(* IEC 61131-3 sources: AXOpen/src/components.cognex.vision/app/SystemConstants (part 2) *)

(* ---- plc_main_IoAddresses.st ---- *)
CONFIGURATION IoAddresses
    VAR_GLOBAL
        CommunicationCard_Engine_Control_1_InputAddress AT %IL1288: LWORD;
        CommunicationCard_Engine_Control_1_OutputAddress AT %QB1267: BYTE;
        CommunicationCard_Engine_Control_2_InputAddress AT %IL1280: LWORD;
        CommunicationCard_Engine_Control_2_OutputAddress AT %QB1266: BYTE;
        CommunicationCard_Engine_Control_3_InputAddress AT %IL1272: LWORD;
        CommunicationCard_Engine_Control_3_OutputAddress AT %QB1265: BYTE;
        CommunicationCard_Engine_Control_4_InputAddress AT %IL1264: LWORD;
        CommunicationCard_Engine_Control_4_OutputAddress AT %QB1264: BYTE;
        CommunicationCard_Result_Data_240_bytes_1_InputAddress_0 AT %IL1024: LWORD;
        CommunicationCard_Result_Data_240_bytes_1_InputAddress_1 AT %IL1032: LWORD;
        CommunicationCard_Result_Data_240_bytes_1_InputAddress_2 AT %IL1040: LWORD;
        CommunicationCard_Result_Data_240_bytes_1_InputAddress_3 AT %IL1048: LWORD;
        CommunicationCard_Result_Data_240_bytes_1_InputAddress_4 AT %IL1056: LWORD;
        CommunicationCard_Result_Data_240_bytes_1_InputAddress_5 AT %IL1064: LWORD;
        CommunicationCard_Result_Data_240_bytes_1_InputAddress_6 AT %IL1072: LWORD;
        CommunicationCard_Result_Data_240_bytes_1_InputAddress_7 AT %IL1080: LWORD;
        CommunicationCard_Result_Data_240_bytes_1_InputAddress_8 AT %IL1088: LWORD;
        CommunicationCard_Result_Data_240_bytes_1_InputAddress_9 AT %IL1096: LWORD;
        CommunicationCard_Result_Data_240_bytes_1_InputAddress_10 AT %IL1104: LWORD;
        CommunicationCard_Result_Data_240_bytes_1_InputAddress_11 AT %IL1112: LWORD;
        CommunicationCard_Result_Data_240_bytes_1_InputAddress_12 AT %IL1120: LWORD;
        CommunicationCard_Result_Data_240_bytes_1_InputAddress_13 AT %IL1128: LWORD;
        CommunicationCard_Result_Data_240_bytes_1_InputAddress_14 AT %IL1136: LWORD;
        CommunicationCard_Result_Data_240_bytes_1_InputAddress_15 AT %IL1144: LWORD;
        CommunicationCard_Result_Data_240_bytes_1_InputAddress_16 AT %IL1152: LWORD;
        CommunicationCard_Result_Data_240_bytes_1_InputAddress_17 AT %IL1160: LWORD;
        CommunicationCard_Result_Data_240_bytes_1_InputAddress_18 AT %IL1168: LWORD;
        CommunicationCard_Result_Data_240_bytes_1_InputAddress_19 AT %IL1176: LWORD;
        CommunicationCard_Result_Data_240_bytes_1_InputAddress_20 AT %IL1184: LWORD;
        CommunicationCard_Result_Data_240_bytes_1_InputAddress_21 AT %IL1192: LWORD;
        CommunicationCard_Result_Data_240_bytes_1_InputAddress_22 AT %IL1200: LWORD;
        CommunicationCard_Result_Data_240_bytes_1_InputAddress_23 AT %IL1208: LWORD;
        CommunicationCard_Result_Data_240_bytes_1_InputAddress_24 AT %IL1216: LWORD;
        CommunicationCard_Result_Data_240_bytes_1_InputAddress_25 AT %IL1224: LWORD;
        CommunicationCard_Result_Data_240_bytes_1_InputAddress_26 AT %IL1232: LWORD;
        CommunicationCard_Result_Data_240_bytes_1_InputAddress_27 AT %IL1240: LWORD;
        CommunicationCard_Result_Data_240_bytes_1_InputAddress_28 AT %IL1248: LWORD;
        CommunicationCard_Result_Data_240_bytes_1_InputAddress_29 AT %IL1256: LWORD;
        CommunicationCard_Result_Data_240_bytes_2_InputAddress_0 AT %IL784: LWORD;
        CommunicationCard_Result_Data_240_bytes_2_InputAddress_1 AT %IL792: LWORD;
        CommunicationCard_Result_Data_240_bytes_2_InputAddress_2 AT %IL800: LWORD;
        CommunicationCard_Result_Data_240_bytes_2_InputAddress_3 AT %IL808: LWORD;
        CommunicationCard_Result_Data_240_bytes_2_InputAddress_4 AT %IL816: LWORD;
        CommunicationCard_Result_Data_240_bytes_2_InputAddress_5 AT %IL824: LWORD;
        CommunicationCard_Result_Data_240_bytes_2_InputAddress_6 AT %IL832: LWORD;
        CommunicationCard_Result_Data_240_bytes_2_InputAddress_7 AT %IL840: LWORD;
        CommunicationCard_Result_Data_240_bytes_2_InputAddress_8 AT %IL848: LWORD;
        CommunicationCard_Result_Data_240_bytes_2_InputAddress_9 AT %IL856: LWORD;
        CommunicationCard_Result_Data_240_bytes_2_InputAddress_10 AT %IL864: LWORD;
        CommunicationCard_Result_Data_240_bytes_2_InputAddress_11 AT %IL872: LWORD;
        CommunicationCard_Result_Data_240_bytes_2_InputAddress_12 AT %IL880: LWORD;
        CommunicationCard_Result_Data_240_bytes_2_InputAddress_13 AT %IL888: LWORD;
        CommunicationCard_Result_Data_240_bytes_2_InputAddress_14 AT %IL896: LWORD;
        CommunicationCard_Result_Data_240_bytes_2_InputAddress_15 AT %IL904: LWORD;
        CommunicationCard_Result_Data_240_bytes_2_InputAddress_16 AT %IL912: LWORD;
        CommunicationCard_Result_Data_240_bytes_2_InputAddress_17 AT %IL920: LWORD;
        CommunicationCard_Result_Data_240_bytes_2_InputAddress_18 AT %IL928: LWORD;
        CommunicationCard_Result_Data_240_bytes_2_InputAddress_19 AT %IL936: LWORD;
        CommunicationCard_Result_Data_240_bytes_2_InputAddress_20 AT %IL944: LWORD;
        CommunicationCard_Result_Data_240_bytes_2_InputAddress_21 AT %IL952: LWORD;
        CommunicationCard_Result_Data_240_bytes_2_InputAddress_22 AT %IL960: LWORD;
        CommunicationCard_Result_Data_240_bytes_2_InputAddress_23 AT %IL968: LWORD;
        CommunicationCard_Result_Data_240_bytes_2_InputAddress_24 AT %IL976: LWORD;
        CommunicationCard_Result_Data_240_bytes_2_InputAddress_25 AT %IL984: LWORD;
        CommunicationCard_Result_Data_240_bytes_2_InputAddress_26 AT %IL992: LWORD;
        CommunicationCard_Result_Data_240_bytes_2_InputAddress_27 AT %IL1000: LWORD;
        CommunicationCard_Result_Data_240_bytes_2_InputAddress_28 AT %IL1008: LWORD;
        CommunicationCard_Result_Data_240_bytes_2_InputAddress_29 AT %IL1016: LWORD;
        CommunicationCard_Result_Data_240_bytes_3_InputAddress_0 AT %IL544: LWORD;
        CommunicationCard_Result_Data_240_bytes_3_InputAddress_1 AT %IL552: LWORD;
        CommunicationCard_Result_Data_240_bytes_3_InputAddress_2 AT %IL560: LWORD;
        CommunicationCard_Result_Data_240_bytes_3_InputAddress_3 AT %IL568: LWORD;
        CommunicationCard_Result_Data_240_bytes_3_InputAddress_4 AT %IL576: LWORD;
        CommunicationCard_Result_Data_240_bytes_3_InputAddress_5 AT %IL584: LWORD;
        CommunicationCard_Result_Data_240_bytes_3_InputAddress_6 AT %IL592: LWORD;
        CommunicationCard_Result_Data_240_bytes_3_InputAddress_7 AT %IL600: LWORD;
        CommunicationCard_Result_Data_240_bytes_3_InputAddress_8 AT %IL608: LWORD;
        CommunicationCard_Result_Data_240_bytes_3_InputAddress_9 AT %IL616: LWORD;
        CommunicationCard_Result_Data_240_bytes_3_InputAddress_10 AT %IL624: LWORD;
        CommunicationCard_Result_Data_240_bytes_3_InputAddress_11 AT %IL632: LWORD;
        CommunicationCard_Result_Data_240_bytes_3_InputAddress_12 AT %IL640: LWORD;
        CommunicationCard_Result_Data_240_bytes_3_InputAddress_13 AT %IL648: LWORD;
        CommunicationCard_Result_Data_240_bytes_3_InputAddress_14 AT %IL656: LWORD;
        CommunicationCard_Result_Data_240_bytes_3_InputAddress_15 AT %IL664: LWORD;
        CommunicationCard_Result_Data_240_bytes_3_InputAddress_16 AT %IL672: LWORD;
        CommunicationCard_Result_Data_240_bytes_3_InputAddress_17 AT %IL680: LWORD;
        CommunicationCard_Result_Data_240_bytes_3_InputAddress_18 AT %IL688: LWORD;
        CommunicationCard_Result_Data_240_bytes_3_InputAddress_19 AT %IL696: LWORD;
        CommunicationCard_Result_Data_240_bytes_3_InputAddress_20 AT %IL704: LWORD;
        CommunicationCard_Result_Data_240_bytes_3_InputAddress_21 AT %IL712: LWORD;
        CommunicationCard_Result_Data_240_bytes_3_InputAddress_22 AT %IL720: LWORD;
        CommunicationCard_Result_Data_240_bytes_3_InputAddress_23 AT %IL728: LWORD;
        CommunicationCard_Result_Data_240_bytes_3_InputAddress_24 AT %IL736: LWORD;
        CommunicationCard_Result_Data_240_bytes_3_InputAddress_25 AT %IL744: LWORD;
        CommunicationCard_Result_Data_240_bytes_3_InputAddress_26 AT %IL752: LWORD;
        CommunicationCard_Result_Data_240_bytes_3_InputAddress_27 AT %IL760: LWORD;
        CommunicationCard_Result_Data_240_bytes_3_InputAddress_28 AT %IL768: LWORD;
        CommunicationCard_Result_Data_240_bytes_3_InputAddress_29 AT %IL776: LWORD;
        CommunicationCard_Result_Data_240_bytes_4_InputAddress_0 AT %IL304: LWORD;
        CommunicationCard_Result_Data_240_bytes_4_InputAddress_1 AT %IL312: LWORD;
        CommunicationCard_Result_Data_240_bytes_4_InputAddress_2 AT %IL320: LWORD;
        CommunicationCard_Result_Data_240_bytes_4_InputAddress_3 AT %IL328: LWORD;
        CommunicationCard_Result_Data_240_bytes_4_InputAddress_4 AT %IL336: LWORD;
        CommunicationCard_Result_Data_240_bytes_4_InputAddress_5 AT %IL344: LWORD;
        CommunicationCard_Result_Data_240_bytes_4_InputAddress_6 AT %IL352: LWORD;
        CommunicationCard_Result_Data_240_bytes_4_InputAddress_7 AT %IL360: LWORD;
        CommunicationCard_Result_Data_240_bytes_4_InputAddress_8 AT %IL368: LWORD;
        CommunicationCard_Result_Data_240_bytes_4_InputAddress_9 AT %IL376: LWORD;
        CommunicationCard_Result_Data_240_bytes_4_InputAddress_10 AT %IL384: LWORD;
        CommunicationCard_Result_Data_240_bytes_4_InputAddress_11 AT %IL392: LWORD;
        CommunicationCard_Result_Data_240_bytes_4_InputAddress_12 AT %IL400: LWORD;
        CommunicationCard_Result_Data_240_bytes_4_InputAddress_13 AT %IL408: LWORD;
        CommunicationCard_Result_Data_240_bytes_4_InputAddress_14 AT %IL416: LWORD;
        CommunicationCard_Result_Data_240_bytes_4_InputAddress_15 AT %IL424: LWORD;
        CommunicationCard_Result_Data_240_bytes_4_InputAddress_16 AT %IL432: LWORD;
        CommunicationCard_Result_Data_240_bytes_4_InputAddress_17 AT %IL440: LWORD;
        CommunicationCard_Result_Data_240_bytes_4_InputAddress_18 AT %IL448: LWORD;
        CommunicationCard_Result_Data_240_bytes_4_InputAddress_19 AT %IL456: LWORD;
        CommunicationCard_Result_Data_240_bytes_4_InputAddress_20 AT %IL464: LWORD;
        CommunicationCard_Result_Data_240_bytes_4_InputAddress_21 AT %IL472: LWORD;
        CommunicationCard_Result_Data_240_bytes_4_InputAddress_22 AT %IL480: LWORD;
        CommunicationCard_Result_Data_240_bytes_4_InputAddress_23 AT %IL488: LWORD;
        CommunicationCard_Result_Data_240_bytes_4_InputAddress_24 AT %IL496: LWORD;
        CommunicationCard_Result_Data_240_bytes_4_InputAddress_25 AT %IL504: LWORD;
        CommunicationCard_Result_Data_240_bytes_4_InputAddress_26 AT %IL512: LWORD;
        CommunicationCard_Result_Data_240_bytes_4_InputAddress_27 AT %IL520: LWORD;
        CommunicationCard_Result_Data_240_bytes_4_InputAddress_28 AT %IL528: LWORD;
        CommunicationCard_Result_Data_240_bytes_4_InputAddress_29 AT %IL536: LWORD;
        CommunicationCard_Result_Data_240_bytes_5_InputAddress_0 AT %IL64: LWORD;
        CommunicationCard_Result_Data_240_bytes_5_InputAddress_1 AT %IL72: LWORD;
        CommunicationCard_Result_Data_240_bytes_5_InputAddress_2 AT %IL80: LWORD;
        CommunicationCard_Result_Data_240_bytes_5_InputAddress_3 AT %IL88: LWORD;
        CommunicationCard_Result_Data_240_bytes_5_InputAddress_4 AT %IL96: LWORD;
        CommunicationCard_Result_Data_240_bytes_5_InputAddress_5 AT %IL104: LWORD;
        CommunicationCard_Result_Data_240_bytes_5_InputAddress_6 AT %IL112: LWORD;
        CommunicationCard_Result_Data_240_bytes_5_InputAddress_7 AT %IL120: LWORD;
        CommunicationCard_Result_Data_240_bytes_5_InputAddress_8 AT %IL128: LWORD;
        CommunicationCard_Result_Data_240_bytes_5_InputAddress_9 AT %IL136: LWORD;
        CommunicationCard_Result_Data_240_bytes_5_InputAddress_10 AT %IL144: LWORD;
        CommunicationCard_Result_Data_240_bytes_5_InputAddress_11 AT %IL152: LWORD;
        CommunicationCard_Result_Data_240_bytes_5_InputAddress_12 AT %IL160: LWORD;
        CommunicationCard_Result_Data_240_bytes_5_InputAddress_13 AT %IL168: LWORD;
        CommunicationCard_Result_Data_240_bytes_5_InputAddress_14 AT %IL176: LWORD;
        CommunicationCard_Result_Data_240_bytes_5_InputAddress_15 AT %IL184: LWORD;
        CommunicationCard_Result_Data_240_bytes_5_InputAddress_16 AT %IL192: LWORD;
        CommunicationCard_Result_Data_240_bytes_5_InputAddress_17 AT %IL200: LWORD;
        CommunicationCard_Result_Data_240_bytes_5_InputAddress_18 AT %IL208: LWORD;
        CommunicationCard_Result_Data_240_bytes_5_InputAddress_19 AT %IL216: LWORD;
        CommunicationCard_Result_Data_240_bytes_5_InputAddress_20 AT %IL224: LWORD;
        CommunicationCard_Result_Data_240_bytes_5_InputAddress_21 AT %IL232: LWORD;
        CommunicationCard_Result_Data_240_bytes_5_InputAddress_22 AT %IL240: LWORD;
        CommunicationCard_Result_Data_240_bytes_5_InputAddress_23 AT %IL248: LWORD;
        CommunicationCard_Result_Data_240_bytes_5_InputAddress_24 AT %IL256: LWORD;
        CommunicationCard_Result_Data_240_bytes_5_InputAddress_25 AT %IL264: LWORD;
        CommunicationCard_Result_Data_240_bytes_5_InputAddress_26 AT %IL272: LWORD;
        CommunicationCard_Result_Data_240_bytes_5_InputAddress_27 AT %IL280: LWORD;
        CommunicationCard_Result_Data_240_bytes_5_InputAddress_28 AT %IL288: LWORD;
        CommunicationCard_Result_Data_240_bytes_5_InputAddress_29 AT %IL296: LWORD;
        CommunicationCard_Result_Data_64_bytes_1_InputAddress_0 AT %IL0: LWORD;
        CommunicationCard_Result_Data_64_bytes_1_InputAddress_1 AT %IL8: LWORD;
        CommunicationCard_Result_Data_64_bytes_1_InputAddress_2 AT %IL16: LWORD;
        CommunicationCard_Result_Data_64_bytes_1_InputAddress_3 AT %IL24: LWORD;
        CommunicationCard_Result_Data_64_bytes_1_InputAddress_4 AT %IL32: LWORD;
        CommunicationCard_Result_Data_64_bytes_1_InputAddress_5 AT %IL40: LWORD;
        CommunicationCard_Result_Data_64_bytes_1_InputAddress_6 AT %IL48: LWORD;
        CommunicationCard_Result_Data_64_bytes_1_InputAddress_7 AT %IL56: LWORD;
        CommunicationCard_System_Control_InputAddress_0 AT %IL1296: LWORD;
        CommunicationCard_System_Control_InputAddress_1 AT %IL1304: LWORD;
        CommunicationCard_System_Control_OutputAddress_0 AT %QL1268: LWORD;
        CommunicationCard_System_Control_OutputAddress_1 AT %QL1276: LWORD;
        CommunicationCard_User_Data_240_bytes_1_OutputAddress_0 AT %QL1024: LWORD;
        CommunicationCard_User_Data_240_bytes_1_OutputAddress_1 AT %QL1032: LWORD;
        CommunicationCard_User_Data_240_bytes_1_OutputAddress_2 AT %QL1040: LWORD;
        CommunicationCard_User_Data_240_bytes_1_OutputAddress_3 AT %QL1048: LWORD;
        CommunicationCard_User_Data_240_bytes_1_OutputAddress_4 AT %QL1056: LWORD;
        CommunicationCard_User_Data_240_bytes_1_OutputAddress_5 AT %QL1064: LWORD;
        CommunicationCard_User_Data_240_bytes_1_OutputAddress_6 AT %QL1072: LWORD;
        CommunicationCard_User_Data_240_bytes_1_OutputAddress_7 AT %QL1080: LWORD;
        CommunicationCard_User_Data_240_bytes_1_OutputAddress_8 AT %QL1088: LWORD;
        CommunicationCard_User_Data_240_bytes_1_OutputAddress_9 AT %QL1096: LWORD;
        CommunicationCard_User_Data_240_bytes_1_OutputAddress_10 AT %QL1104: LWORD;
        CommunicationCard_User_Data_240_bytes_1_OutputAddress_11 AT %QL1112: LWORD;
        CommunicationCard_User_Data_240_bytes_1_OutputAddress_12 AT %QL1120: LWORD;
        CommunicationCard_User_Data_240_bytes_1_OutputAddress_13 AT %QL1128: LWORD;
        CommunicationCard_User_Data_240_bytes_1_OutputAddress_14 AT %QL1136: LWORD;
        CommunicationCard_User_Data_240_bytes_1_OutputAddress_15 AT %QL1144: LWORD;
        CommunicationCard_User_Data_240_bytes_1_OutputAddress_16 AT %QL1152: LWORD;
        CommunicationCard_User_Data_240_bytes_1_OutputAddress_17 AT %QL1160: LWORD;
        CommunicationCard_User_Data_240_bytes_1_OutputAddress_18 AT %QL1168: LWORD;
        CommunicationCard_User_Data_240_bytes_1_OutputAddress_19 AT %QL1176: LWORD;
        CommunicationCard_User_Data_240_bytes_1_OutputAddress_20 AT %QL1184: LWORD;
        CommunicationCard_User_Data_240_bytes_1_OutputAddress_21 AT %QL1192: LWORD;
        CommunicationCard_User_Data_240_bytes_1_OutputAddress_22 AT %QL1200: LWORD;
        CommunicationCard_User_Data_240_bytes_1_OutputAddress_23 AT %QL1208: LWORD;
        CommunicationCard_User_Data_240_bytes_1_OutputAddress_24 AT %QL1216: LWORD;
        CommunicationCard_User_Data_240_bytes_1_OutputAddress_25 AT %QL1224: LWORD;
        CommunicationCard_User_Data_240_bytes_1_OutputAddress_26 AT %QL1232: LWORD;
        CommunicationCard_User_Data_240_bytes_1_OutputAddress_27 AT %QL1240: LWORD;
        CommunicationCard_User_Data_240_bytes_1_OutputAddress_28 AT %QL1248: LWORD;
        CommunicationCard_User_Data_240_bytes_1_OutputAddress_29 AT %QL1256: LWORD;
        CommunicationCard_User_Data_240_bytes_2_OutputAddress_0 AT %QL784: LWORD;
        CommunicationCard_User_Data_240_bytes_2_OutputAddress_1 AT %QL792: LWORD;
        CommunicationCard_User_Data_240_bytes_2_OutputAddress_2 AT %QL800: LWORD;
        CommunicationCard_User_Data_240_bytes_2_OutputAddress_3 AT %QL808: LWORD;
        CommunicationCard_User_Data_240_bytes_2_OutputAddress_4 AT %QL816: LWORD;
        CommunicationCard_User_Data_240_bytes_2_OutputAddress_5 AT %QL824: LWORD;
        CommunicationCard_User_Data_240_bytes_2_OutputAddress_6 AT %QL832: LWORD;
        CommunicationCard_User_Data_240_bytes_2_OutputAddress_7 AT %QL840: LWORD;
        CommunicationCard_User_Data_240_bytes_2_OutputAddress_8 AT %QL848: LWORD;
        CommunicationCard_User_Data_240_bytes_2_OutputAddress_9 AT %QL856: LWORD;
        CommunicationCard_User_Data_240_bytes_2_OutputAddress_10 AT %QL864: LWORD;
        CommunicationCard_User_Data_240_bytes_2_OutputAddress_11 AT %QL872: LWORD;
        CommunicationCard_User_Data_240_bytes_2_OutputAddress_12 AT %QL880: LWORD;
        CommunicationCard_User_Data_240_bytes_2_OutputAddress_13 AT %QL888: LWORD;
        CommunicationCard_User_Data_240_bytes_2_OutputAddress_14 AT %QL896: LWORD;
        CommunicationCard_User_Data_240_bytes_2_OutputAddress_15 AT %QL904: LWORD;
        CommunicationCard_User_Data_240_bytes_2_OutputAddress_16 AT %QL912: LWORD;
        CommunicationCard_User_Data_240_bytes_2_OutputAddress_17 AT %QL920: LWORD;
        CommunicationCard_User_Data_240_bytes_2_OutputAddress_18 AT %QL928: LWORD;
        CommunicationCard_User_Data_240_bytes_2_OutputAddress_19 AT %QL936: LWORD;
        CommunicationCard_User_Data_240_bytes_2_OutputAddress_20 AT %QL944: LWORD;
        CommunicationCard_User_Data_240_bytes_2_OutputAddress_21 AT %QL952: LWORD;
        CommunicationCard_User_Data_240_bytes_2_OutputAddress_22 AT %QL960: LWORD;
        CommunicationCard_User_Data_240_bytes_2_OutputAddress_23 AT %QL968: LWORD;
        CommunicationCard_User_Data_240_bytes_2_OutputAddress_24 AT %QL976: LWORD;
        CommunicationCard_User_Data_240_bytes_2_OutputAddress_25 AT %QL984: LWORD;
        CommunicationCard_User_Data_240_bytes_2_OutputAddress_26 AT %QL992: LWORD;
        CommunicationCard_User_Data_240_bytes_2_OutputAddress_27 AT %QL1000: LWORD;
        CommunicationCard_User_Data_240_bytes_2_OutputAddress_28 AT %QL1008: LWORD;
        CommunicationCard_User_Data_240_bytes_2_OutputAddress_29 AT %QL1016: LWORD;
        CommunicationCard_User_Data_240_bytes_3_OutputAddress_0 AT %QL544: LWORD;
        CommunicationCard_User_Data_240_bytes_3_OutputAddress_1 AT %QL552: LWORD;
        CommunicationCard_User_Data_240_bytes_3_OutputAddress_2 AT %QL560: LWORD;
        CommunicationCard_User_Data_240_bytes_3_OutputAddress_3 AT %QL568: LWORD;
        CommunicationCard_User_Data_240_bytes_3_OutputAddress_4 AT %QL576: LWORD;
        CommunicationCard_User_Data_240_bytes_3_OutputAddress_5 AT %QL584: LWORD;
        CommunicationCard_User_Data_240_bytes_3_OutputAddress_6 AT %QL592: LWORD;
        CommunicationCard_User_Data_240_bytes_3_OutputAddress_7 AT %QL600: LWORD;
        CommunicationCard_User_Data_240_bytes_3_OutputAddress_8 AT %QL608: LWORD;
        CommunicationCard_User_Data_240_bytes_3_OutputAddress_9 AT %QL616: LWORD;
        CommunicationCard_User_Data_240_bytes_3_OutputAddress_10 AT %QL624: LWORD;
        CommunicationCard_User_Data_240_bytes_3_OutputAddress_11 AT %QL632: LWORD;
        CommunicationCard_User_Data_240_bytes_3_OutputAddress_12 AT %QL640: LWORD;
        CommunicationCard_User_Data_240_bytes_3_OutputAddress_13 AT %QL648: LWORD;
        CommunicationCard_User_Data_240_bytes_3_OutputAddress_14 AT %QL656: LWORD;
        CommunicationCard_User_Data_240_bytes_3_OutputAddress_15 AT %QL664: LWORD;
        CommunicationCard_User_Data_240_bytes_3_OutputAddress_16 AT %QL672: LWORD;
        CommunicationCard_User_Data_240_bytes_3_OutputAddress_17 AT %QL680: LWORD;
        CommunicationCard_User_Data_240_bytes_3_OutputAddress_18 AT %QL688: LWORD;
        CommunicationCard_User_Data_240_bytes_3_OutputAddress_19 AT %QL696: LWORD;
        CommunicationCard_User_Data_240_bytes_3_OutputAddress_20 AT %QL704: LWORD;
        CommunicationCard_User_Data_240_bytes_3_OutputAddress_21 AT %QL712: LWORD;
        CommunicationCard_User_Data_240_bytes_3_OutputAddress_22 AT %QL720: LWORD;
        CommunicationCard_User_Data_240_bytes_3_OutputAddress_23 AT %QL728: LWORD;
        CommunicationCard_User_Data_240_bytes_3_OutputAddress_24 AT %QL736: LWORD;
        CommunicationCard_User_Data_240_bytes_3_OutputAddress_25 AT %QL744: LWORD;
        CommunicationCard_User_Data_240_bytes_3_OutputAddress_26 AT %QL752: LWORD;
        CommunicationCard_User_Data_240_bytes_3_OutputAddress_27 AT %QL760: LWORD;
        CommunicationCard_User_Data_240_bytes_3_OutputAddress_28 AT %QL768: LWORD;
        CommunicationCard_User_Data_240_bytes_3_OutputAddress_29 AT %QL776: LWORD;
        CommunicationCard_User_Data_240_bytes_4_OutputAddress_0 AT %QL304: LWORD;
        CommunicationCard_User_Data_240_bytes_4_OutputAddress_1 AT %QL312: LWORD;
        CommunicationCard_User_Data_240_bytes_4_OutputAddress_2 AT %QL320: LWORD;
        CommunicationCard_User_Data_240_bytes_4_OutputAddress_3 AT %QL328: LWORD;
        CommunicationCard_User_Data_240_bytes_4_OutputAddress_4 AT %QL336: LWORD;
        CommunicationCard_User_Data_240_bytes_4_OutputAddress_5 AT %QL344: LWORD;
        CommunicationCard_User_Data_240_bytes_4_OutputAddress_6 AT %QL352: LWORD;
        CommunicationCard_User_Data_240_bytes_4_OutputAddress_7 AT %QL360: LWORD;
        CommunicationCard_User_Data_240_bytes_4_OutputAddress_8 AT %QL368: LWORD;
        CommunicationCard_User_Data_240_bytes_4_OutputAddress_9 AT %QL376: LWORD;
        CommunicationCard_User_Data_240_bytes_4_OutputAddress_10 AT %QL384: LWORD;
        CommunicationCard_User_Data_240_bytes_4_OutputAddress_11 AT %QL392: LWORD;
        CommunicationCard_User_Data_240_bytes_4_OutputAddress_12 AT %QL400: LWORD;
        CommunicationCard_User_Data_240_bytes_4_OutputAddress_13 AT %QL408: LWORD;
        CommunicationCard_User_Data_240_bytes_4_OutputAddress_14 AT %QL416: LWORD;
        CommunicationCard_User_Data_240_bytes_4_OutputAddress_15 AT %QL424: LWORD;
        CommunicationCard_User_Data_240_bytes_4_OutputAddress_16 AT %QL432: LWORD;
        CommunicationCard_User_Data_240_bytes_4_OutputAddress_17 AT %QL440: LWORD;
        CommunicationCard_User_Data_240_bytes_4_OutputAddress_18 AT %QL448: LWORD;
        CommunicationCard_User_Data_240_bytes_4_OutputAddress_19 AT %QL456: LWORD;
        CommunicationCard_User_Data_240_bytes_4_OutputAddress_20 AT %QL464: LWORD;
        CommunicationCard_User_Data_240_bytes_4_OutputAddress_21 AT %QL472: LWORD;
        CommunicationCard_User_Data_240_bytes_4_OutputAddress_22 AT %QL480: LWORD;
        CommunicationCard_User_Data_240_bytes_4_OutputAddress_23 AT %QL488: LWORD;
        CommunicationCard_User_Data_240_bytes_4_OutputAddress_24 AT %QL496: LWORD;
        CommunicationCard_User_Data_240_bytes_4_OutputAddress_25 AT %QL504: LWORD;
        CommunicationCard_User_Data_240_bytes_4_OutputAddress_26 AT %QL512: LWORD;
        CommunicationCard_User_Data_240_bytes_4_OutputAddress_27 AT %QL520: LWORD;
        CommunicationCard_User_Data_240_bytes_4_OutputAddress_28 AT %QL528: LWORD;
        CommunicationCard_User_Data_240_bytes_4_OutputAddress_29 AT %QL536: LWORD;
        CommunicationCard_User_Data_240_bytes_5_OutputAddress_0 AT %QL64: LWORD;
        CommunicationCard_User_Data_240_bytes_5_OutputAddress_1 AT %QL72: LWORD;
        CommunicationCard_User_Data_240_bytes_5_OutputAddress_2 AT %QL80: LWORD;
        CommunicationCard_User_Data_240_bytes_5_OutputAddress_3 AT %QL88: LWORD;
        CommunicationCard_User_Data_240_bytes_5_OutputAddress_4 AT %QL96: LWORD;
        CommunicationCard_User_Data_240_bytes_5_OutputAddress_5 AT %QL104: LWORD;
        CommunicationCard_User_Data_240_bytes_5_OutputAddress_6 AT %QL112: LWORD;
        CommunicationCard_User_Data_240_bytes_5_OutputAddress_7 AT %QL120: LWORD;
        CommunicationCard_User_Data_240_bytes_5_OutputAddress_8 AT %QL128: LWORD;
        CommunicationCard_User_Data_240_bytes_5_OutputAddress_9 AT %QL136: LWORD;
        CommunicationCard_User_Data_240_bytes_5_OutputAddress_10 AT %QL144: LWORD;
        CommunicationCard_User_Data_240_bytes_5_OutputAddress_11 AT %QL152: LWORD;
        CommunicationCard_User_Data_240_bytes_5_OutputAddress_12 AT %QL160: LWORD;
        CommunicationCard_User_Data_240_bytes_5_OutputAddress_13 AT %QL168: LWORD;
        CommunicationCard_User_Data_240_bytes_5_OutputAddress_14 AT %QL176: LWORD;
        CommunicationCard_User_Data_240_bytes_5_OutputAddress_15 AT %QL184: LWORD;
        CommunicationCard_User_Data_240_bytes_5_OutputAddress_16 AT %QL192: LWORD;
        CommunicationCard_User_Data_240_bytes_5_OutputAddress_17 AT %QL200: LWORD;
        CommunicationCard_User_Data_240_bytes_5_OutputAddress_18 AT %QL208: LWORD;
        CommunicationCard_User_Data_240_bytes_5_OutputAddress_19 AT %QL216: LWORD;
        CommunicationCard_User_Data_240_bytes_5_OutputAddress_20 AT %QL224: LWORD;
        CommunicationCard_User_Data_240_bytes_5_OutputAddress_21 AT %QL232: LWORD;
        CommunicationCard_User_Data_240_bytes_5_OutputAddress_22 AT %QL240: LWORD;
        CommunicationCard_User_Data_240_bytes_5_OutputAddress_23 AT %QL248: LWORD;
        CommunicationCard_User_Data_240_bytes_5_OutputAddress_24 AT %QL256: LWORD;
        CommunicationCard_User_Data_240_bytes_5_OutputAddress_25 AT %QL264: LWORD;
        CommunicationCard_User_Data_240_bytes_5_OutputAddress_26 AT %QL272: LWORD;
        CommunicationCard_User_Data_240_bytes_5_OutputAddress_27 AT %QL280: LWORD;
        CommunicationCard_User_Data_240_bytes_5_OutputAddress_28 AT %QL288: LWORD;
        CommunicationCard_User_Data_240_bytes_5_OutputAddress_29 AT %QL296: LWORD;
        CommunicationCard_User_Data_64_bytes_1_OutputAddress_0 AT %QL0: LWORD;
        CommunicationCard_User_Data_64_bytes_1_OutputAddress_1 AT %QL8: LWORD;
        CommunicationCard_User_Data_64_bytes_1_OutputAddress_2 AT %QL16: LWORD;
        CommunicationCard_User_Data_64_bytes_1_OutputAddress_3 AT %QL24: LWORD;
        CommunicationCard_User_Data_64_bytes_1_OutputAddress_4 AT %QL32: LWORD;
        CommunicationCard_User_Data_64_bytes_1_OutputAddress_5 AT %QL40: LWORD;
        CommunicationCard_User_Data_64_bytes_1_OutputAddress_6 AT %QL48: LWORD;
        CommunicationCard_User_Data_64_bytes_1_OutputAddress_7 AT %QL56: LWORD;
        st10_dm280_Acquisition_Control_OutputAddress AT %QB1487: BYTE;
        st10_dm280_Acquisition_Status_InputAddress_0 AT %IB1527: BYTE;
        st10_dm280_Acquisition_Status_InputAddress_1 AT %IB1528: BYTE;
        st10_dm280_Acquisition_Status_InputAddress_2 AT %IB1529: BYTE;
        st10_dm280_Result_Data_128_bytes_InputAddress_0 AT %IL1390: LWORD;
        st10_dm280_Result_Data_128_bytes_InputAddress_1 AT %IL1398: LWORD;
        st10_dm280_Result_Data_128_bytes_InputAddress_2 AT %IL1406: LWORD;
        st10_dm280_Result_Data_128_bytes_InputAddress_3 AT %IL1414: LWORD;
        st10_dm280_Result_Data_128_bytes_InputAddress_4 AT %IL1422: LWORD;
        st10_dm280_Result_Data_128_bytes_InputAddress_5 AT %IL1430: LWORD;
        st10_dm280_Result_Data_128_bytes_InputAddress_6 AT %IL1438: LWORD;
        st10_dm280_Result_Data_128_bytes_InputAddress_7 AT %IL1446: LWORD;
        st10_dm280_Result_Data_128_bytes_InputAddress_8 AT %IL1454: LWORD;
        st10_dm280_Result_Data_128_bytes_InputAddress_9 AT %IL1462: LWORD;
        st10_dm280_Result_Data_128_bytes_InputAddress_10 AT %IL1470: LWORD;
        st10_dm280_Result_Data_128_bytes_InputAddress_11 AT %IL1478: LWORD;
        st10_dm280_Result_Data_128_bytes_InputAddress_12 AT %IL1486: LWORD;
        st10_dm280_Result_Data_128_bytes_InputAddress_13 AT %IL1494: LWORD;
        st10_dm280_Result_Data_128_bytes_InputAddress_14 AT %IL1502: LWORD;
        st10_dm280_Result_Data_128_bytes_InputAddress_15 AT %IL1510: LWORD;
        st10_dm280_Result_Data_128_bytes_InputAddress_16 AT %IL1518: LWORD;
        st10_dm280_Results_Control_OutputAddress AT %QB1486: BYTE;
        st10_dm280_Results_Status_InputAddress AT %IB1526: BYTE;
        st10_dm280_Soft_Event_Control_InputAddress AT %IB1530: BYTE;
        st10_dm280_Soft_Event_Control_OutputAddress AT %QB1485: BYTE;
        st10_dm280_User_Data_128_bytes_OutputAddress_0 AT %QD1353: DWORD;
        st10_dm280_User_Data_128_bytes_OutputAddress_1 AT %QD1357: DWORD;
        st10_dm280_User_Data_128_bytes_OutputAddress_2 AT %QD1361: DWORD;
        st10_dm280_User_Data_128_bytes_OutputAddress_3 AT %QD1365: DWORD;
        st10_dm280_User_Data_128_bytes_OutputAddress_4 AT %QD1369: DWORD;
        st10_dm280_User_Data_128_bytes_OutputAddress_5 AT %QD1373: DWORD;
        st10_dm280_User_Data_128_bytes_OutputAddress_6 AT %QD1377: DWORD;
        st10_dm280_User_Data_128_bytes_OutputAddress_7 AT %QD1381: DWORD;
        st10_dm280_User_Data_128_bytes_OutputAddress_8 AT %QD1385: DWORD;
        st10_dm280_User_Data_128_bytes_OutputAddress_9 AT %QD1389: DWORD;
        st10_dm280_User_Data_128_bytes_OutputAddress_10 AT %QD1393: DWORD;
        st10_dm280_User_Data_128_bytes_OutputAddress_11 AT %QD1397: DWORD;
        st10_dm280_User_Data_128_bytes_OutputAddress_12 AT %QD1401: DWORD;
        st10_dm280_User_Data_128_bytes_OutputAddress_13 AT %QD1405: DWORD;
        st10_dm280_User_Data_128_bytes_OutputAddress_14 AT %QD1409: DWORD;
        st10_dm280_User_Data_128_bytes_OutputAddress_15 AT %QD1413: DWORD;
        st10_dm280_User_Data_128_bytes_OutputAddress_16 AT %QD1417: DWORD;
        st10_dm280_User_Data_128_bytes_OutputAddress_17 AT %QD1421: DWORD;
        st10_dm280_User_Data_128_bytes_OutputAddress_18 AT %QD1425: DWORD;
        st10_dm280_User_Data_128_bytes_OutputAddress_19 AT %QD1429: DWORD;
        st10_dm280_User_Data_128_bytes_OutputAddress_20 AT %QD1433: DWORD;
        st10_dm280_User_Data_128_bytes_OutputAddress_21 AT %QD1437: DWORD;
        st10_dm280_User_Data_128_bytes_OutputAddress_22 AT %QD1441: DWORD;
        st10_dm280_User_Data_128_bytes_OutputAddress_23 AT %QD1445: DWORD;
        st10_dm280_User_Data_128_bytes_OutputAddress_24 AT %QD1449: DWORD;
        st10_dm280_User_Data_128_bytes_OutputAddress_25 AT %QD1453: DWORD;
        st10_dm280_User_Data_128_bytes_OutputAddress_26 AT %QD1457: DWORD;
        st10_dm280_User_Data_128_bytes_OutputAddress_27 AT %QD1461: DWORD;
        st10_dm280_User_Data_128_bytes_OutputAddress_28 AT %QD1465: DWORD;
        st10_dm280_User_Data_128_bytes_OutputAddress_29 AT %QD1469: DWORD;
        st10_dm280_User_Data_128_bytes_OutputAddress_30 AT %QD1473: DWORD;
        st10_dm280_User_Data_128_bytes_OutputAddress_31 AT %QD1477: DWORD;
        st10_dm280_User_Data_128_bytes_OutputAddress_32 AT %QD1481: DWORD;
        st10_is2802m_Acquisition_Control_OutputAddress AT %QB2508: BYTE;
        st10_is2802m_Acquisition_Status_InputAddress AT %ID2535: DWORD;
        st10_is2802m_Command_Control_InputAddress AT %ID2543: DWORD;
        st10_is2802m_Command_Control_OutputAddress AT %QW2504: WORD;
        st10_is2802m_Inspection_Control_OutputAddress AT %QB2507: BYTE;
        st10_is2802m_Inspection_Status_InputAddress AT %ID2539: DWORD;
        st10_is2802m_Result_Data_250_bytes_1_InputAddress_0 AT %IW2281: WORD;
        st10_is2802m_Result_Data_250_bytes_1_InputAddress_1 AT %IW2283: WORD;
        st10_is2802m_Result_Data_250_bytes_1_InputAddress_2 AT %IW2285: WORD;
        st10_is2802m_Result_Data_250_bytes_1_InputAddress_3 AT %IW2287: WORD;
        st10_is2802m_Result_Data_250_bytes_1_InputAddress_4 AT %IW2289: WORD;
        st10_is2802m_Result_Data_250_bytes_1_InputAddress_5 AT %IW2291: WORD;
        st10_is2802m_Result_Data_250_bytes_1_InputAddress_6 AT %IW2293: WORD;
        st10_is2802m_Result_Data_250_bytes_1_InputAddress_7 AT %IW2295: WORD;
        st10_is2802m_Result_Data_250_bytes_1_InputAddress_8 AT %IW2297: WORD;
        st10_is2802m_Result_Data_250_bytes_1_InputAddress_9 AT %IW2299: WORD;
        st10_is2802m_Result_Data_250_bytes_1_InputAddress_10 AT %IW2301: WORD;
        st10_is2802m_Result_Data_250_bytes_1_InputAddress_11 AT %IW2303: WORD;
        st10_is2802m_Result_Data_250_bytes_1_InputAddress_12 AT %IW2305: WORD;
        st10_is2802m_Result_Data_250_bytes_1_InputAddress_13 AT %IW2307: WORD;
        st10_is2802m_Result_Data_250_bytes_1_InputAddress_14 AT %IW2309: WORD;
        st10_is2802m_Result_Data_250_bytes_1_InputAddress_15 AT %IW2311: WORD;
        st10_is2802m_Result_Data_250_bytes_1_InputAddress_16 AT %IW2313: WORD;
        st10_is2802m_Result_Data_250_bytes_1_InputAddress_17 AT %IW2315: WORD;
        st10_is2802m_Result_Data_250_bytes_1_InputAddress_18 AT %IW2317: WORD;
        st10_is2802m_Result_Data_250_bytes_1_InputAddress_19 AT %IW2319: WORD;
        st10_is2802m_Result_Data_250_bytes_1_InputAddress_20 AT %IW2321: WORD;
        st10_is2802m_Result_Data_250_bytes_1_InputAddress_21 AT %IW2323: WORD;
        st10_is2802m_Result_Data_250_bytes_1_InputAddress_22 AT %IW2325: WORD;
        st10_is2802m_Result_Data_250_bytes_1_InputAddress_23 AT %IW2327: WORD;
        st10_is2802m_Result_Data_250_bytes_1_InputAddress_24 AT %IW2329: WORD;
        st10_is2802m_Result_Data_250_bytes_1_InputAddress_25 AT %IW2331: WORD;
        st10_is2802m_Result_Data_250_bytes_1_InputAddress_26 AT %IW2333: WORD;
        st10_is2802m_Result_Data_250_bytes_1_InputAddress_27 AT %IW2335: WORD;
        st10_is2802m_Result_Data_250_bytes_1_InputAddress_28 AT %IW2337: WORD;
        st10_is2802m_Result_Data_250_bytes_1_InputAddress_29 AT %IW2339: WORD;
        st10_is2802m_Result_Data_250_bytes_1_InputAddress_30 AT %IW2341: WORD;
        st10_is2802m_Result_Data_250_bytes_1_InputAddress_31 AT %IW2343: WORD;
        st10_is2802m_Result_Data_250_bytes_1_InputAddress_32 AT %IW2345: WORD;
        st10_is2802m_Result_Data_250_bytes_1_InputAddress_33 AT %IW2347: WORD;
        st10_is2802m_Result_Data_250_bytes_1_InputAddress_34 AT %IW2349: WORD;
        st10_is2802m_Result_Data_250_bytes_1_InputAddress_35 AT %IW2351: WORD;
        st10_is2802m_Result_Data_250_bytes_1_InputAddress_36 AT %IW2353: WORD;
        st10_is2802m_Result_Data_250_bytes_1_InputAddress_37 AT %IW2355: WORD;
        st10_is2802m_Result_Data_250_bytes_1_InputAddress_38 AT %IW2357: WORD;
        st10_is2802m_Result_Data_250_bytes_1_InputAddress_39 AT %IW2359: WORD;
        st10_is2802m_Result_Data_250_bytes_1_InputAddress_40 AT %IW2361: WORD;
        st10_is2802m_Result_Data_250_bytes_1_InputAddress_41 AT %IW2363: WORD;
        st10_is2802m_Result_Data_250_bytes_1_InputAddress_42 AT %IW2365: WORD;
        st10_is2802m_Result_Data_250_bytes_1_InputAddress_43 AT %IW2367: WORD;
        st10_is2802m_Result_Data_250_bytes_1_InputAddress_44 AT %IW2369: WORD;
        st10_is2802m_Result_Data_250_bytes_1_InputAddress_45 AT %IW2371: WORD;
        st10_is2802m_Result_Data_250_bytes_1_InputAddress_46 AT %IW2373: WORD;
        st10_is2802m_Result_Data_250_bytes_1_InputAddress_47 AT %IW2375: WORD;
        st10_is2802m_Result_Data_250_bytes_1_InputAddress_48 AT %IW2377: WORD;
        st10_is2802m_Result_Data_250_bytes_1_InputAddress_49 AT %IW2379: WORD;
        st10_is2802m_Result_Data_250_bytes_1_InputAddress_50 AT %IW2381: WORD;
        st10_is2802m_Result_Data_250_bytes_1_InputAddress_51 AT %IW2383: WORD;
        st10_is2802m_Result_Data_250_bytes_1_InputAddress_52 AT %IW2385: WORD;
        st10_is2802m_Result_Data_250_bytes_1_InputAddress_53 AT %IW2387: WORD;
        st10_is2802m_Result_Data_250_bytes_1_InputAddress_54 AT %IW2389: WORD;
        st10_is2802m_Result_Data_250_bytes_1_InputAddress_55 AT %IW2391: WORD;
        st10_is2802m_Result_Data_250_bytes_1_InputAddress_56 AT %IW2393: WORD;
        st10_is2802m_Result_Data_250_bytes_1_InputAddress_57 AT %IW2395: WORD;
        st10_is2802m_Result_Data_250_bytes_1_InputAddress_58 AT %IW2397: WORD;
        st10_is2802m_Result_Data_250_bytes_1_InputAddress_59 AT %IW2399: WORD;
        st10_is2802m_Result_Data_250_bytes_1_InputAddress_60 AT %IW2401: WORD;
        st10_is2802m_Result_Data_250_bytes_1_InputAddress_61 AT %IW2403: WORD;
        st10_is2802m_Result_Data_250_bytes_1_InputAddress_62 AT %IW2405: WORD;
        st10_is2802m_Result_Data_250_bytes_1_InputAddress_63 AT %IW2407: WORD;
        st10_is2802m_Result_Data_250_bytes_1_InputAddress_64 AT %IW2409: WORD;
        st10_is2802m_Result_Data_250_bytes_1_InputAddress_65 AT %IW2411: WORD;
        st10_is2802m_Result_Data_250_bytes_1_InputAddress_66 AT %IW2413: WORD;
        st10_is2802m_Result_Data_250_bytes_1_InputAddress_67 AT %IW2415: WORD;
        st10_is2802m_Result_Data_250_bytes_1_InputAddress_68 AT %IW2417: WORD;
        st10_is2802m_Result_Data_250_bytes_1_InputAddress_69 AT %IW2419: WORD;
        st10_is2802m_Result_Data_250_bytes_1_InputAddress_70 AT %IW2421: WORD;
        st10_is2802m_Result_Data_250_bytes_1_InputAddress_71 AT %IW2423: WORD;
        st10_is2802m_Result_Data_250_bytes_1_InputAddress_72 AT %IW2425: WORD;
        st10_is2802m_Result_Data_250_bytes_1_InputAddress_73 AT %IW2427: WORD;
        st10_is2802m_Result_Data_250_bytes_1_InputAddress_74 AT %IW2429: WORD;
        st10_is2802m_Result_Data_250_bytes_1_InputAddress_75 AT %IW2431: WORD;
        st10_is2802m_Result_Data_250_bytes_1_InputAddress_76 AT %IW2433: WORD;
        st10_is2802m_Result_Data_250_bytes_1_InputAddress_77 AT %IW2435: WORD;
        st10_is2802m_Result_Data_250_bytes_1_InputAddress_78 AT %IW2437: WORD;
        st10_is2802m_Result_Data_250_bytes_1_InputAddress_79 AT %IW2439: WORD;
        st10_is2802m_Result_Data_250_bytes_1_InputAddress_80 AT %IW2441: WORD;
        st10_is2802m_Result_Data_250_bytes_1_InputAddress_81 AT %IW2443: WORD;
        st10_is2802m_Result_Data_250_bytes_1_InputAddress_82 AT %IW2445: WORD;
        st10_is2802m_Result_Data_250_bytes_1_InputAddress_83 AT %IW2447: WORD;
        st10_is2802m_Result_Data_250_bytes_1_InputAddress_84 AT %IW2449: WORD;
        st10_is2802m_Result_Data_250_bytes_1_InputAddress_85 AT %IW2451: WORD;
        st10_is2802m_Result_Data_250_bytes_1_InputAddress_86 AT %IW2453: WORD;
        st10_is2802m_Result_Data_250_bytes_1_InputAddress_87 AT %IW2455: WORD;
        st10_is2802m_Result_Data_250_bytes_1_InputAddress_88 AT %IW2457: WORD;
        st10_is2802m_Result_Data_250_bytes_1_InputAddress_89 AT %IW2459: WORD;
        st10_is2802m_Result_Data_250_bytes_1_InputAddress_90 AT %IW2461: WORD;
        st10_is2802m_Result_Data_250_bytes_1_InputAddress_91 AT %IW2463: WORD;
        st10_is2802m_Result_Data_250_bytes_1_InputAddress_92 AT %IW2465: WORD;
        st10_is2802m_Result_Data_250_bytes_1_InputAddress_93 AT %IW2467: WORD;
        st10_is2802m_Result_Data_250_bytes_1_InputAddress_94 AT %IW2469: WORD;
        st10_is2802m_Result_Data_250_bytes_1_InputAddress_95 AT %IW2471: WORD;
        st10_is2802m_Result_Data_250_bytes_1_InputAddress_96 AT %IW2473: WORD;
        st10_is2802m_Result_Data_250_bytes_1_InputAddress_97 AT %IW2475: WORD;
        st10_is2802m_Result_Data_250_bytes_1_InputAddress_98 AT %IW2477: WORD;
        st10_is2802m_Result_Data_250_bytes_1_InputAddress_99 AT %IW2479: WORD;
        st10_is2802m_Result_Data_250_bytes_1_InputAddress_100 AT %IW2481: WORD;
        st10_is2802m_Result_Data_250_bytes_1_InputAddress_101 AT %IW2483: WORD;
        st10_is2802m_Result_Data_250_bytes_1_InputAddress_102 AT %IW2485: WORD;
        st10_is2802m_Result_Data_250_bytes_1_InputAddress_103 AT %IW2487: WORD;
        st10_is2802m_Result_Data_250_bytes_1_InputAddress_104 AT %IW2489: WORD;
        st10_is2802m_Result_Data_250_bytes_1_InputAddress_105 AT %IW2491: WORD;
        st10_is2802m_Result_Data_250_bytes_1_InputAddress_106 AT %IW2493: WORD;
        st10_is2802m_Result_Data_250_bytes_1_InputAddress_107 AT %IW2495: WORD;
        st10_is2802m_Result_Data_250_bytes_1_InputAddress_108 AT %IW2497: WORD;
        st10_is2802m_Result_Data_250_bytes_1_InputAddress_109 AT %IW2499: WORD;
        st10_is2802m_Result_Data_250_bytes_1_InputAddress_110 AT %IW2501: WORD;
        st10_is2802m_Result_Data_250_bytes_1_InputAddress_111 AT %IW2503: WORD;
        st10_is2802m_Result_Data_250_bytes_1_InputAddress_112 AT %IW2505: WORD;
        st10_is2802m_Result_Data_250_bytes_1_InputAddress_113 AT %IW2507: WORD;
        st10_is2802m_Result_Data_250_bytes_1_InputAddress_114 AT %IW2509: WORD;
        st10_is2802m_Result_Data_250_bytes_1_InputAddress_115 AT %IW2511: WORD;
        st10_is2802m_Result_Data_250_bytes_1_InputAddress_116 AT %IW2513: WORD;
        st10_is2802m_Result_Data_250_bytes_1_InputAddress_117 AT %IW2515: WORD;
        st10_is2802m_Result_Data_250_bytes_1_InputAddress_118 AT %IW2517: WORD;
        st10_is2802m_Result_Data_250_bytes_1_InputAddress_119 AT %IW2519: WORD;
        st10_is2802m_Result_Data_250_bytes_1_InputAddress_120 AT %IW2521: WORD;
        st10_is2802m_Result_Data_250_bytes_1_InputAddress_121 AT %IW2523: WORD;
        st10_is2802m_Result_Data_250_bytes_1_InputAddress_122 AT %IW2525: WORD;
        st10_is2802m_Result_Data_250_bytes_1_InputAddress_123 AT %IW2527: WORD;
        st10_is2802m_Result_Data_250_bytes_1_InputAddress_124 AT %IW2529: WORD;
        st10_is2802m_Result_Data_250_bytes_1_InputAddress_125 AT %IW2531: WORD;
        st10_is2802m_Result_Data_250_bytes_1_InputAddress_126 AT %IW2533: WORD;
        st10_is2802m_Result_Data_250_bytes_2_InputAddress_0 AT %IW2031: WORD;
        st10_is2802m_Result_Data_250_bytes_2_InputAddress_1 AT %IW2033: WORD;
        st10_is2802m_Result_Data_250_bytes_2_InputAddress_2 AT %IW2035: WORD;
        st10_is2802m_Result_Data_250_bytes_2_InputAddress_3 AT %IW2037: WORD;
        st10_is2802m_Result_Data_250_bytes_2_InputAddress_4 AT %IW2039: WORD;
        st10_is2802m_Result_Data_250_bytes_2_InputAddress_5 AT %IW2041: WORD;
        st10_is2802m_Result_Data_250_bytes_2_InputAddress_6 AT %IW2043: WORD;
        st10_is2802m_Result_Data_250_bytes_2_InputAddress_7 AT %IW2045: WORD;
        st10_is2802m_Result_Data_250_bytes_2_InputAddress_8 AT %IW2047: WORD;
        st10_is2802m_Result_Data_250_bytes_2_InputAddress_9 AT %IW2049: WORD;
        st10_is2802m_Result_Data_250_bytes_2_InputAddress_10 AT %IW2051: WORD;
        st10_is2802m_Result_Data_250_bytes_2_InputAddress_11 AT %IW2053: WORD;
        st10_is2802m_Result_Data_250_bytes_2_InputAddress_12 AT %IW2055: WORD;
        st10_is2802m_Result_Data_250_bytes_2_InputAddress_13 AT %IW2057: WORD;
        st10_is2802m_Result_Data_250_bytes_2_InputAddress_14 AT %IW2059: WORD;
        st10_is2802m_Result_Data_250_bytes_2_InputAddress_15 AT %IW2061: WORD;
        st10_is2802m_Result_Data_250_bytes_2_InputAddress_16 AT %IW2063: WORD;
        st10_is2802m_Result_Data_250_bytes_2_InputAddress_17 AT %IW2065: WORD;
        st10_is2802m_Result_Data_250_bytes_2_InputAddress_18 AT %IW2067: WORD;
        st10_is2802m_Result_Data_250_bytes_2_InputAddress_19 AT %IW2069: WORD;
        st10_is2802m_Result_Data_250_bytes_2_InputAddress_20 AT %IW2071: WORD;
        st10_is2802m_Result_Data_250_bytes_2_InputAddress_21 AT %IW2073: WORD;
        st10_is2802m_Result_Data_250_bytes_2_InputAddress_22 AT %IW2075: WORD;
        st10_is2802m_Result_Data_250_bytes_2_InputAddress_23 AT %IW2077: WORD;
        st10_is2802m_Result_Data_250_bytes_2_InputAddress_24 AT %IW2079: WORD;
        st10_is2802m_Result_Data_250_bytes_2_InputAddress_25 AT %IW2081: WORD;
        st10_is2802m_Result_Data_250_bytes_2_InputAddress_26 AT %IW2083: WORD;
        st10_is2802m_Result_Data_250_bytes_2_InputAddress_27 AT %IW2085: WORD;
        st10_is2802m_Result_Data_250_bytes_2_InputAddress_28 AT %IW2087: WORD;
        st10_is2802m_Result_Data_250_bytes_2_InputAddress_29 AT %IW2089: WORD;
        st10_is2802m_Result_Data_250_bytes_2_InputAddress_30 AT %IW2091: WORD;
        st10_is2802m_Result_Data_250_bytes_2_InputAddress_31 AT %IW2093: WORD;
        st10_is2802m_Result_Data_250_bytes_2_InputAddress_32 AT %IW2095: WORD;
        st10_is2802m_Result_Data_250_bytes_2_InputAddress_33 AT %IW2097: WORD;
        st10_is2802m_Result_Data_250_bytes_2_InputAddress_34 AT %IW2099: WORD;
        st10_is2802m_Result_Data_250_bytes_2_InputAddress_35 AT %IW2101: WORD;
        st10_is2802m_Result_Data_250_bytes_2_InputAddress_36 AT %IW2103: WORD;
        st10_is2802m_Result_Data_250_bytes_2_InputAddress_37 AT %IW2105: WORD;
        st10_is2802m_Result_Data_250_bytes_2_InputAddress_38 AT %IW2107: WORD;
        st10_is2802m_Result_Data_250_bytes_2_InputAddress_39 AT %IW2109: WORD;
        st10_is2802m_Result_Data_250_bytes_2_InputAddress_40 AT %IW2111: WORD;
        st10_is2802m_Result_Data_250_bytes_2_InputAddress_41 AT %IW2113: WORD;
        st10_is2802m_Result_Data_250_bytes_2_InputAddress_42 AT %IW2115: WORD;
        st10_is2802m_Result_Data_250_bytes_2_InputAddress_43 AT %IW2117: WORD;
        st10_is2802m_Result_Data_250_bytes_2_InputAddress_44 AT %IW2119: WORD;
        st10_is2802m_Result_Data_250_bytes_2_InputAddress_45 AT %IW2121: WORD;
        st10_is2802m_Result_Data_250_bytes_2_InputAddress_46 AT %IW2123: WORD;
        st10_is2802m_Result_Data_250_bytes_2_InputAddress_47 AT %IW2125: WORD;
        st10_is2802m_Result_Data_250_bytes_2_InputAddress_48 AT %IW2127: WORD;
        st10_is2802m_Result_Data_250_bytes_2_InputAddress_49 AT %IW2129: WORD;
        st10_is2802m_Result_Data_250_bytes_2_InputAddress_50 AT %IW2131: WORD;
        st10_is2802m_Result_Data_250_bytes_2_InputAddress_51 AT %IW2133: WORD;
        st10_is2802m_Result_Data_250_bytes_2_InputAddress_52 AT %IW2135: WORD;
        st10_is2802m_Result_Data_250_bytes_2_InputAddress_53 AT %IW2137: WORD;
        st10_is2802m_Result_Data_250_bytes_2_InputAddress_54 AT %IW2139: WORD;
        st10_is2802m_Result_Data_250_bytes_2_InputAddress_55 AT %IW2141: WORD;
        st10_is2802m_Result_Data_250_bytes_2_InputAddress_56 AT %IW2143: WORD;
        st10_is2802m_Result_Data_250_bytes_2_InputAddress_57 AT %IW2145: WORD;
        st10_is2802m_Result_Data_250_bytes_2_InputAddress_58 AT %IW2147: WORD;
        st10_is2802m_Result_Data_250_bytes_2_InputAddress_59 AT %IW2149: WORD;
        st10_is2802m_Result_Data_250_bytes_2_InputAddress_60 AT %IW2151: WORD;
        st10_is2802m_Result_Data_250_bytes_2_InputAddress_61 AT %IW2153: WORD;
        st10_is2802m_Result_Data_250_bytes_2_InputAddress_62 AT %IW2155: WORD;
        st10_is2802m_Result_Data_250_bytes_2_InputAddress_63 AT %IW2157: WORD;
        st10_is2802m_Result_Data_250_bytes_2_InputAddress_64 AT %IW2159: WORD;
        st10_is2802m_Result_Data_250_bytes_2_InputAddress_65 AT %IW2161: WORD;
        st10_is2802m_Result_Data_250_bytes_2_InputAddress_66 AT %IW2163: WORD;
        st10_is2802m_Result_Data_250_bytes_2_InputAddress_67 AT %IW2165: WORD;
        st10_is2802m_Result_Data_250_bytes_2_InputAddress_68 AT %IW2167: WORD;
        st10_is2802m_Result_Data_250_bytes_2_InputAddress_69 AT %IW2169: WORD;
        st10_is2802m_Result_Data_250_bytes_2_InputAddress_70 AT %IW2171: WORD;
        st10_is2802m_Result_Data_250_bytes_2_InputAddress_71 AT %IW2173: WORD;
        st10_is2802m_Result_Data_250_bytes_2_InputAddress_72 AT %IW2175: WORD;
        st10_is2802m_Result_Data_250_bytes_2_InputAddress_73 AT %IW2177: WORD;
        st10_is2802m_Result_Data_250_bytes_2_InputAddress_74 AT %IW2179: WORD;
        st10_is2802m_Result_Data_250_bytes_2_InputAddress_75 AT %IW2181: WORD;
        st10_is2802m_Result_Data_250_bytes_2_InputAddress_76 AT %IW2183: WORD;
        st10_is2802m_Result_Data_250_bytes_2_InputAddress_77 AT %IW2185: WORD;
        st10_is2802m_Result_Data_250_bytes_2_InputAddress_78 AT %IW2187: WORD;
        st10_is2802m_Result_Data_250_bytes_2_InputAddress_79 AT %IW2189: WORD;
        st10_is2802m_Result_Data_250_bytes_2_InputAddress_80 AT %IW2191: WORD;
        st10_is2802m_Result_Data_250_bytes_2_InputAddress_81 AT %IW2193: WORD;
        st10_is2802m_Result_Data_250_bytes_2_InputAddress_82 AT %IW2195: WORD;
        st10_is2802m_Result_Data_250_bytes_2_InputAddress_83 AT %IW2197: WORD;
        st10_is2802m_Result_Data_250_bytes_2_InputAddress_84 AT %IW2199: WORD;
        st10_is2802m_Result_Data_250_bytes_2_InputAddress_85 AT %IW2201: WORD;
        st10_is2802m_Result_Data_250_bytes_2_InputAddress_86 AT %IW2203: WORD;
        st10_is2802m_Result_Data_250_bytes_2_InputAddress_87 AT %IW2205: WORD;
        st10_is2802m_Result_Data_250_bytes_2_InputAddress_88 AT %IW2207: WORD;
        st10_is2802m_Result_Data_250_bytes_2_InputAddress_89 AT %IW2209: WORD;
        st10_is2802m_Result_Data_250_bytes_2_InputAddress_90 AT %IW2211: WORD;
        st10_is2802m_Result_Data_250_bytes_2_InputAddress_91 AT %IW2213: WORD;
        st10_is2802m_Result_Data_250_bytes_2_InputAddress_92 AT %IW2215: WORD;
        st10_is2802m_Result_Data_250_bytes_2_InputAddress_93 AT %IW2217: WORD;
        st10_is2802m_Result_Data_250_bytes_2_InputAddress_94 AT %IW2219: WORD;
        st10_is2802m_Result_Data_250_bytes_2_InputAddress_95 AT %IW2221: WORD;
        st10_is2802m_Result_Data_250_bytes_2_InputAddress_96 AT %IW2223: WORD;
        st10_is2802m_Result_Data_250_bytes_2_InputAddress_97 AT %IW2225: WORD;
        st10_is2802m_Result_Data_250_bytes_2_InputAddress_98 AT %IW2227: WORD;
        st10_is2802m_Result_Data_250_bytes_2_InputAddress_99 AT %IW2229: WORD;
        st10_is2802m_Result_Data_250_bytes_2_InputAddress_100 AT %IW2231: WORD;
        st10_is2802m_Result_Data_250_bytes_2_InputAddress_101 AT %IW2233: WORD;
        st10_is2802m_Result_Data_250_bytes_2_InputAddress_102 AT %IW2235: WORD;
        st10_is2802m_Result_Data_250_bytes_2_InputAddress_103 AT %IW2237: WORD;
        st10_is2802m_Result_Data_250_bytes_2_InputAddress_104 AT %IW2239: WORD;
        st10_is2802m_Result_Data_250_bytes_2_InputAddress_105 AT %IW2241: WORD;
        st10_is2802m_Result_Data_250_bytes_2_InputAddress_106 AT %IW2243: WORD;
        st10_is2802m_Result_Data_250_bytes_2_InputAddress_107 AT %IW2245: WORD;
        st10_is2802m_Result_Data_250_bytes_2_InputAddress_108 AT %IW2247: WORD;
        st10_is2802m_Result_Data_250_bytes_2_InputAddress_109 AT %IW2249: WORD;
        st10_is2802m_Result_Data_250_bytes_2_InputAddress_110 AT %IW2251: WORD;
        st10_is2802m_Result_Data_250_bytes_2_InputAddress_111 AT %IW2253: WORD;
        st10_is2802m_Result_Data_250_bytes_2_InputAddress_112 AT %IW2255: WORD;
        st10_is2802m_Result_Data_250_bytes_2_InputAddress_113 AT %IW2257: WORD;
        st10_is2802m_Result_Data_250_bytes_2_InputAddress_114 AT %IW2259: WORD;
        st10_is2802m_Result_Data_250_bytes_2_InputAddress_115 AT %IW2261: WORD;
        st10_is2802m_Result_Data_250_bytes_2_InputAddress_116 AT %IW2263: WORD;
        st10_is2802m_Result_Data_250_bytes_2_InputAddress_117 AT %IW2265: WORD;
        st10_is2802m_Result_Data_250_bytes_2_InputAddress_118 AT %IW2267: WORD;
        st10_is2802m_Result_Data_250_bytes_2_InputAddress_119 AT %IW2269: WORD;
        st10_is2802m_Result_Data_250_bytes_2_InputAddress_120 AT %IW2271: WORD;
        st10_is2802m_Result_Data_250_bytes_2_InputAddress_121 AT %IW2273: WORD;
        st10_is2802m_Result_Data_250_bytes_2_InputAddress_122 AT %IW2275: WORD;
        st10_is2802m_Result_Data_250_bytes_2_InputAddress_123 AT %IW2277: WORD;
        st10_is2802m_Result_Data_250_bytes_2_InputAddress_124 AT %IW2279: WORD;
        st10_is2802m_Result_Data_250_bytes_3_InputAddress_0 AT %IW1781: WORD;
        st10_is2802m_Result_Data_250_bytes_3_InputAddress_1 AT %IW1783: WORD;
        st10_is2802m_Result_Data_250_bytes_3_InputAddress_2 AT %IW1785: WORD;
        st10_is2802m_Result_Data_250_bytes_3_InputAddress_3 AT %IW1787: WORD;
        st10_is2802m_Result_Data_250_bytes_3_InputAddress_4 AT %IW1789: WORD;
        st10_is2802m_Result_Data_250_bytes_3_InputAddress_5 AT %IW1791: WORD;
        st10_is2802m_Result_Data_250_bytes_3_InputAddress_6 AT %IW1793: WORD;
        st10_is2802m_Result_Data_250_bytes_3_InputAddress_7 AT %IW1795: WORD;
        st10_is2802m_Result_Data_250_bytes_3_InputAddress_8 AT %IW1797: WORD;
        st10_is2802m_Result_Data_250_bytes_3_InputAddress_9 AT %IW1799: WORD;
        st10_is2802m_Result_Data_250_bytes_3_InputAddress_10 AT %IW1801: WORD;
        st10_is2802m_Result_Data_250_bytes_3_InputAddress_11 AT %IW1803: WORD;
        st10_is2802m_Result_Data_250_bytes_3_InputAddress_12 AT %IW1805: WORD;
        st10_is2802m_Result_Data_250_bytes_3_InputAddress_13 AT %IW1807: WORD;
        st10_is2802m_Result_Data_250_bytes_3_InputAddress_14 AT %IW1809: WORD;
        st10_is2802m_Result_Data_250_bytes_3_InputAddress_15 AT %IW1811: WORD;
        st10_is2802m_Result_Data_250_bytes_3_InputAddress_16 AT %IW1813: WORD;
        st10_is2802m_Result_Data_250_bytes_3_InputAddress_17 AT %IW1815: WORD;
        st10_is2802m_Result_Data_250_bytes_3_InputAddress_18 AT %IW1817: WORD;
        st10_is2802m_Result_Data_250_bytes_3_InputAddress_19 AT %IW1819: WORD;
        st10_is2802m_Result_Data_250_bytes_3_InputAddress_20 AT %IW1821: WORD;
        st10_is2802m_Result_Data_250_bytes_3_InputAddress_21 AT %IW1823: WORD;
        st10_is2802m_Result_Data_250_bytes_3_InputAddress_22 AT %IW1825: WORD;
        st10_is2802m_Result_Data_250_bytes_3_InputAddress_23 AT %IW1827: WORD;
        st10_is2802m_Result_Data_250_bytes_3_InputAddress_24 AT %IW1829: WORD;
        st10_is2802m_Result_Data_250_bytes_3_InputAddress_25 AT %IW1831: WORD;
        st10_is2802m_Result_Data_250_bytes_3_InputAddress_26 AT %IW1833: WORD;
        st10_is2802m_Result_Data_250_bytes_3_InputAddress_27 AT %IW1835: WORD;
        st10_is2802m_Result_Data_250_bytes_3_InputAddress_28 AT %IW1837: WORD;
        st10_is2802m_Result_Data_250_bytes_3_InputAddress_29 AT %IW1839: WORD;
        st10_is2802m_Result_Data_250_bytes_3_InputAddress_30 AT %IW1841: WORD;
        st10_is2802m_Result_Data_250_bytes_3_InputAddress_31 AT %IW1843: WORD;
        st10_is2802m_Result_Data_250_bytes_3_InputAddress_32 AT %IW1845: WORD;
        st10_is2802m_Result_Data_250_bytes_3_InputAddress_33 AT %IW1847: WORD;
        st10_is2802m_Result_Data_250_bytes_3_InputAddress_34 AT %IW1849: WORD;
        st10_is2802m_Result_Data_250_bytes_3_InputAddress_35 AT %IW1851: WORD;
        st10_is2802m_Result_Data_250_bytes_3_InputAddress_36 AT %IW1853: WORD;
        st10_is2802m_Result_Data_250_bytes_3_InputAddress_37 AT %IW1855: WORD;
        st10_is2802m_Result_Data_250_bytes_3_InputAddress_38 AT %IW1857: WORD;
        st10_is2802m_Result_Data_250_bytes_3_InputAddress_39 AT %IW1859: WORD;
        st10_is2802m_Result_Data_250_bytes_3_InputAddress_40 AT %IW1861: WORD;
        st10_is2802m_Result_Data_250_bytes_3_InputAddress_41 AT %IW1863: WORD;
        st10_is2802m_Result_Data_250_bytes_3_InputAddress_42 AT %IW1865: WORD;
        st10_is2802m_Result_Data_250_bytes_3_InputAddress_43 AT %IW1867: WORD;
        st10_is2802m_Result_Data_250_bytes_3_InputAddress_44 AT %IW1869: WORD;
        st10_is2802m_Result_Data_250_bytes_3_InputAddress_45 AT %IW1871: WORD;
        st10_is2802m_Result_Data_250_bytes_3_InputAddress_46 AT %IW1873: WORD;
        st10_is2802m_Result_Data_250_bytes_3_InputAddress_47 AT %IW1875: WORD;
        st10_is2802m_Result_Data_250_bytes_3_InputAddress_48 AT %IW1877: WORD;
        st10_is2802m_Result_Data_250_bytes_3_InputAddress_49 AT %IW1879: WORD;
        st10_is2802m_Result_Data_250_bytes_3_InputAddress_50 AT %IW1881: WORD;
        st10_is2802m_Result_Data_250_bytes_3_InputAddress_51 AT %IW1883: WORD;
        st10_is2802m_Result_Data_250_bytes_3_InputAddress_52 AT %IW1885: WORD;
        st10_is2802m_Result_Data_250_bytes_3_InputAddress_53 AT %IW1887: WORD;
        st10_is2802m_Result_Data_250_bytes_3_InputAddress_54 AT %IW1889: WORD;
        st10_is2802m_Result_Data_250_bytes_3_InputAddress_55 AT %IW1891: WORD;
        st10_is2802m_Result_Data_250_bytes_3_InputAddress_56 AT %IW1893: WORD;
        st10_is2802m_Result_Data_250_bytes_3_InputAddress_57 AT %IW1895: WORD;
        st10_is2802m_Result_Data_250_bytes_3_InputAddress_58 AT %IW1897: WORD;
        st10_is2802m_Result_Data_250_bytes_3_InputAddress_59 AT %IW1899: WORD;
        st10_is2802m_Result_Data_250_bytes_3_InputAddress_60 AT %IW1901: WORD;
        st10_is2802m_Result_Data_250_bytes_3_InputAddress_61 AT %IW1903: WORD;
        st10_is2802m_Result_Data_250_bytes_3_InputAddress_62 AT %IW1905: WORD;
        st10_is2802m_Result_Data_250_bytes_3_InputAddress_63 AT %IW1907: WORD;
        st10_is2802m_Result_Data_250_bytes_3_InputAddress_64 AT %IW1909: WORD;
        st10_is2802m_Result_Data_250_bytes_3_InputAddress_65 AT %IW1911: WORD;
        st10_is2802m_Result_Data_250_bytes_3_InputAddress_66 AT %IW1913: WORD;
        st10_is2802m_Result_Data_250_bytes_3_InputAddress_67 AT %IW1915: WORD;
        st10_is2802m_Result_Data_250_bytes_3_InputAddress_68 AT %IW1917: WORD;
        st10_is2802m_Result_Data_250_bytes_3_InputAddress_69 AT %IW1919: WORD;
        st10_is2802m_Result_Data_250_bytes_3_InputAddress_70 AT %IW1921: WORD;
        st10_is2802m_Result_Data_250_bytes_3_InputAddress_71 AT %IW1923: WORD;
        st10_is2802m_Result_Data_250_bytes_3_InputAddress_72 AT %IW1925: WORD;
        st10_is2802m_Result_Data_250_bytes_3_InputAddress_73 AT %IW1927: WORD;
        st10_is2802m_Result_Data_250_bytes_3_InputAddress_74 AT %IW1929: WORD;
        st10_is2802m_Result_Data_250_bytes_3_InputAddress_75 AT %IW1931: WORD;
        st10_is2802m_Result_Data_250_bytes_3_InputAddress_76 AT %IW1933: WORD;
        st10_is2802m_Result_Data_250_bytes_3_InputAddress_77 AT %IW1935: WORD;
        st10_is2802m_Result_Data_250_bytes_3_InputAddress_78 AT %IW1937: WORD;
        st10_is2802m_Result_Data_250_bytes_3_InputAddress_79 AT %IW1939: WORD;
        st10_is2802m_Result_Data_250_bytes_3_InputAddress_80 AT %IW1941: WORD;
        st10_is2802m_Result_Data_250_bytes_3_InputAddress_81 AT %IW1943: WORD;
        st10_is2802m_Result_Data_250_bytes_3_InputAddress_82 AT %IW1945: WORD;
        st10_is2802m_Result_Data_250_bytes_3_InputAddress_83 AT %IW1947: WORD;
        st10_is2802m_Result_Data_250_bytes_3_InputAddress_84 AT %IW1949: WORD;
        st10_is2802m_Result_Data_250_bytes_3_InputAddress_85 AT %IW1951: WORD;
        st10_is2802m_Result_Data_250_bytes_3_InputAddress_86 AT %IW1953: WORD;
        st10_is2802m_Result_Data_250_bytes_3_InputAddress_87 AT %IW1955: WORD;
        st10_is2802m_Result_Data_250_bytes_3_InputAddress_88 AT %IW1957: WORD;
        st10_is2802m_Result_Data_250_bytes_3_InputAddress_89 AT %IW1959: WORD;
        st10_is2802m_Result_Data_250_bytes_3_InputAddress_90 AT %IW1961: WORD;
        st10_is2802m_Result_Data_250_bytes_3_InputAddress_91 AT %IW1963: WORD;
        st10_is2802m_Result_Data_250_bytes_3_InputAddress_92 AT %IW1965: WORD;
        st10_is2802m_Result_Data_250_bytes_3_InputAddress_93 AT %IW1967: WORD;
        st10_is2802m_Result_Data_250_bytes_3_InputAddress_94 AT %IW1969: WORD;
        st10_is2802m_Result_Data_250_bytes_3_InputAddress_95 AT %IW1971: WORD;
        st10_is2802m_Result_Data_250_bytes_3_InputAddress_96 AT %IW1973: WORD;
        st10_is2802m_Result_Data_250_bytes_3_InputAddress_97 AT %IW1975: WORD;
        st10_is2802m_Result_Data_250_bytes_3_InputAddress_98 AT %IW1977: WORD;
        st10_is2802m_Result_Data_250_bytes_3_InputAddress_99 AT %IW1979: WORD;
        st10_is2802m_Result_Data_250_bytes_3_InputAddress_100 AT %IW1981: WORD;
        st10_is2802m_Result_Data_250_bytes_3_InputAddress_101 AT %IW1983: WORD;
        st10_is2802m_Result_Data_250_bytes_3_InputAddress_102 AT %IW1985: WORD;
        st10_is2802m_Result_Data_250_bytes_3_InputAddress_103 AT %IW1987: WORD;
        st10_is2802m_Result_Data_250_bytes_3_InputAddress_104 AT %IW1989: WORD;
        st10_is2802m_Result_Data_250_bytes_3_InputAddress_105 AT %IW1991: WORD;
        st10_is2802m_Result_Data_250_bytes_3_InputAddress_106 AT %IW1993: WORD;
        st10_is2802m_Result_Data_250_bytes_3_InputAddress_107 AT %IW1995: WORD;
        st10_is2802m_Result_Data_250_bytes_3_InputAddress_108 AT %IW1997: WORD;
        st10_is2802m_Result_Data_250_bytes_3_InputAddress_109 AT %IW1999: WORD;
        st10_is2802m_Result_Data_250_bytes_3_InputAddress_110 AT %IW2001: WORD;
        st10_is2802m_Result_Data_250_bytes_3_InputAddress_111 AT %IW2003: WORD;
        st10_is2802m_Result_Data_250_bytes_3_InputAddress_112 AT %IW2005: WORD;
        st10_is2802m_Result_Data_250_bytes_3_InputAddress_113 AT %IW2007: WORD;
        st10_is2802m_Result_Data_250_bytes_3_InputAddress_114 AT %IW2009: WORD;
        st10_is2802m_Result_Data_250_bytes_3_InputAddress_115 AT %IW2011: WORD;
        st10_is2802m_Result_Data_250_bytes_3_InputAddress_116 AT %IW2013: WORD;
        st10_is2802m_Result_Data_250_bytes_3_InputAddress_117 AT %IW2015: WORD;
        st10_is2802m_Result_Data_250_bytes_3_InputAddress_118 AT %IW2017: WORD;
        st10_is2802m_Result_Data_250_bytes_3_InputAddress_119 AT %IW2019: WORD;
        st10_is2802m_Result_Data_250_bytes_3_InputAddress_120 AT %IW2021: WORD;
        st10_is2802m_Result_Data_250_bytes_3_InputAddress_121 AT %IW2023: WORD;
        st10_is2802m_Result_Data_250_bytes_3_InputAddress_122 AT %IW2025: WORD;
        st10_is2802m_Result_Data_250_bytes_3_InputAddress_123 AT %IW2027: WORD;
        st10_is2802m_Result_Data_250_bytes_3_InputAddress_124 AT %IW2029: WORD;
        st10_is2802m_Result_Data_250_bytes_4_InputAddress_0 AT %IW1531: WORD;
        st10_is2802m_Result_Data_250_bytes_4_InputAddress_1 AT %IW1533: WORD;
        st10_is2802m_Result_Data_250_bytes_4_InputAddress_2 AT %IW1535: WORD;
        st10_is2802m_Result_Data_250_bytes_4_InputAddress_3 AT %IW1537: WORD;
        st10_is2802m_Result_Data_250_bytes_4_InputAddress_4 AT %IW1539: WORD;
        st10_is2802m_Result_Data_250_bytes_4_InputAddress_5 AT %IW1541: WORD;
        st10_is2802m_Result_Data_250_bytes_4_InputAddress_6 AT %IW1543: WORD;
        st10_is2802m_Result_Data_250_bytes_4_InputAddress_7 AT %IW1545: WORD;
        st10_is2802m_Result_Data_250_bytes_4_InputAddress_8 AT %IW1547: WORD;
        st10_is2802m_Result_Data_250_bytes_4_InputAddress_9 AT %IW1549: WORD;
        st10_is2802m_Result_Data_250_bytes_4_InputAddress_10 AT %IW1551: WORD;
        st10_is2802m_Result_Data_250_bytes_4_InputAddress_11 AT %IW1553: WORD;
        st10_is2802m_Result_Data_250_bytes_4_InputAddress_12 AT %IW1555: WORD;
        st10_is2802m_Result_Data_250_bytes_4_InputAddress_13 AT %IW1557: WORD;
        st10_is2802m_Result_Data_250_bytes_4_InputAddress_14 AT %IW1559: WORD;
        st10_is2802m_Result_Data_250_bytes_4_InputAddress_15 AT %IW1561: WORD;
        st10_is2802m_Result_Data_250_bytes_4_InputAddress_16 AT %IW1563: WORD;
        st10_is2802m_Result_Data_250_bytes_4_InputAddress_17 AT %IW1565: WORD;
        st10_is2802m_Result_Data_250_bytes_4_InputAddress_18 AT %IW1567: WORD;
        st10_is2802m_Result_Data_250_bytes_4_InputAddress_19 AT %IW1569: WORD;
        st10_is2802m_Result_Data_250_bytes_4_InputAddress_20 AT %IW1571: WORD;
        st10_is2802m_Result_Data_250_bytes_4_InputAddress_21 AT %IW1573: WORD;
        st10_is2802m_Result_Data_250_bytes_4_InputAddress_22 AT %IW1575: WORD;
        st10_is2802m_Result_Data_250_bytes_4_InputAddress_23 AT %IW1577: WORD;
        st10_is2802m_Result_Data_250_bytes_4_InputAddress_24 AT %IW1579: WORD;
        st10_is2802m_Result_Data_250_bytes_4_InputAddress_25 AT %IW1581: WORD;
        st10_is2802m_Result_Data_250_bytes_4_InputAddress_26 AT %IW1583: WORD;
        st10_is2802m_Result_Data_250_bytes_4_InputAddress_27 AT %IW1585: WORD;
        st10_is2802m_Result_Data_250_bytes_4_InputAddress_28 AT %IW1587: WORD;
        st10_is2802m_Result_Data_250_bytes_4_InputAddress_29 AT %IW1589: WORD;
        st10_is2802m_Result_Data_250_bytes_4_InputAddress_30 AT %IW1591: WORD;
        st10_is2802m_Result_Data_250_bytes_4_InputAddress_31 AT %IW1593: WORD;
        st10_is2802m_Result_Data_250_bytes_4_InputAddress_32 AT %IW1595: WORD;
        st10_is2802m_Result_Data_250_bytes_4_InputAddress_33 AT %IW1597: WORD;
        st10_is2802m_Result_Data_250_bytes_4_InputAddress_34 AT %IW1599: WORD;
        st10_is2802m_Result_Data_250_bytes_4_InputAddress_35 AT %IW1601: WORD;
        st10_is2802m_Result_Data_250_bytes_4_InputAddress_36 AT %IW1603: WORD;
        st10_is2802m_Result_Data_250_bytes_4_InputAddress_37 AT %IW1605: WORD;
        st10_is2802m_Result_Data_250_bytes_4_InputAddress_38 AT %IW1607: WORD;
        st10_is2802m_Result_Data_250_bytes_4_InputAddress_39 AT %IW1609: WORD;
        st10_is2802m_Result_Data_250_bytes_4_InputAddress_40 AT %IW1611: WORD;
        st10_is2802m_Result_Data_250_bytes_4_InputAddress_41 AT %IW1613: WORD;
        st10_is2802m_Result_Data_250_bytes_4_InputAddress_42 AT %IW1615: WORD;
        st10_is2802m_Result_Data_250_bytes_4_InputAddress_43 AT %IW1617: WORD;
        st10_is2802m_Result_Data_250_bytes_4_InputAddress_44 AT %IW1619: WORD;
        st10_is2802m_Result_Data_250_bytes_4_InputAddress_45 AT %IW1621: WORD;
        st10_is2802m_Result_Data_250_bytes_4_InputAddress_46 AT %IW1623: WORD;
        st10_is2802m_Result_Data_250_bytes_4_InputAddress_47 AT %IW1625: WORD;
        st10_is2802m_Result_Data_250_bytes_4_InputAddress_48 AT %IW1627: WORD;
        st10_is2802m_Result_Data_250_bytes_4_InputAddress_49 AT %IW1629: WORD;
        st10_is2802m_Result_Data_250_bytes_4_InputAddress_50 AT %IW1631: WORD;
        st10_is2802m_Result_Data_250_bytes_4_InputAddress_51 AT %IW1633: WORD;
        st10_is2802m_Result_Data_250_bytes_4_InputAddress_52 AT %IW1635: WORD;
        st10_is2802m_Result_Data_250_bytes_4_InputAddress_53 AT %IW1637: WORD;
        st10_is2802m_Result_Data_250_bytes_4_InputAddress_54 AT %IW1639: WORD;
        st10_is2802m_Result_Data_250_bytes_4_InputAddress_55 AT %IW1641: WORD;
        st10_is2802m_Result_Data_250_bytes_4_InputAddress_56 AT %IW1643: WORD;
        st10_is2802m_Result_Data_250_bytes_4_InputAddress_57 AT %IW1645: WORD;
        st10_is2802m_Result_Data_250_bytes_4_InputAddress_58 AT %IW1647: WORD;
        st10_is2802m_Result_Data_250_bytes_4_InputAddress_59 AT %IW1649: WORD;
        st10_is2802m_Result_Data_250_bytes_4_InputAddress_60 AT %IW1651: WORD;
        st10_is2802m_Result_Data_250_bytes_4_InputAddress_61 AT %IW1653: WORD;
        st10_is2802m_Result_Data_250_bytes_4_InputAddress_62 AT %IW1655: WORD;
        st10_is2802m_Result_Data_250_bytes_4_InputAddress_63 AT %IW1657: WORD;
        st10_is2802m_Result_Data_250_bytes_4_InputAddress_64 AT %IW1659: WORD;
        st10_is2802m_Result_Data_250_bytes_4_InputAddress_65 AT %IW1661: WORD;
        st10_is2802m_Result_Data_250_bytes_4_InputAddress_66 AT %IW1663: WORD;
        st10_is2802m_Result_Data_250_bytes_4_InputAddress_67 AT %IW1665: WORD;
        st10_is2802m_Result_Data_250_bytes_4_InputAddress_68 AT %IW1667: WORD;
        st10_is2802m_Result_Data_250_bytes_4_InputAddress_69 AT %IW1669: WORD;
        st10_is2802m_Result_Data_250_bytes_4_InputAddress_70 AT %IW1671: WORD;
        st10_is2802m_Result_Data_250_bytes_4_InputAddress_71 AT %IW1673: WORD;
        st10_is2802m_Result_Data_250_bytes_4_InputAddress_72 AT %IW1675: WORD;
        st10_is2802m_Result_Data_250_bytes_4_InputAddress_73 AT %IW1677: WORD;
        st10_is2802m_Result_Data_250_bytes_4_InputAddress_74 AT %IW1679: WORD;
        st10_is2802m_Result_Data_250_bytes_4_InputAddress_75 AT %IW1681: WORD;
        st10_is2802m_Result_Data_250_bytes_4_InputAddress_76 AT %IW1683: WORD;
        st10_is2802m_Result_Data_250_bytes_4_InputAddress_77 AT %IW1685: WORD;
        st10_is2802m_Result_Data_250_bytes_4_InputAddress_78 AT %IW1687: WORD;
        st10_is2802m_Result_Data_250_bytes_4_InputAddress_79 AT %IW1689: WORD;
        st10_is2802m_Result_Data_250_bytes_4_InputAddress_80 AT %IW1691: WORD;
        st10_is2802m_Result_Data_250_bytes_4_InputAddress_81 AT %IW1693: WORD;
        st10_is2802m_Result_Data_250_bytes_4_InputAddress_82 AT %IW1695: WORD;
        st10_is2802m_Result_Data_250_bytes_4_InputAddress_83 AT %IW1697: WORD;
        st10_is2802m_Result_Data_250_bytes_4_InputAddress_84 AT %IW1699: WORD;
        st10_is2802m_Result_Data_250_bytes_4_InputAddress_85 AT %IW1701: WORD;
        st10_is2802m_Result_Data_250_bytes_4_InputAddress_86 AT %IW1703: WORD;
        st10_is2802m_Result_Data_250_bytes_4_InputAddress_87 AT %IW1705: WORD;
        st10_is2802m_Result_Data_250_bytes_4_InputAddress_88 AT %IW1707: WORD;
        st10_is2802m_Result_Data_250_bytes_4_InputAddress_89 AT %IW1709: WORD;
        st10_is2802m_Result_Data_250_bytes_4_InputAddress_90 AT %IW1711: WORD;
        st10_is2802m_Result_Data_250_bytes_4_InputAddress_91 AT %IW1713: WORD;
        st10_is2802m_Result_Data_250_bytes_4_InputAddress_92 AT %IW1715: WORD;
        st10_is2802m_Result_Data_250_bytes_4_InputAddress_93 AT %IW1717: WORD;
        st10_is2802m_Result_Data_250_bytes_4_InputAddress_94 AT %IW1719: WORD;
        st10_is2802m_Result_Data_250_bytes_4_InputAddress_95 AT %IW1721: WORD;
        st10_is2802m_Result_Data_250_bytes_4_InputAddress_96 AT %IW1723: WORD;
        st10_is2802m_Result_Data_250_bytes_4_InputAddress_97 AT %IW1725: WORD;
        st10_is2802m_Result_Data_250_bytes_4_InputAddress_98 AT %IW1727: WORD;
        st10_is2802m_Result_Data_250_bytes_4_InputAddress_99 AT %IW1729: WORD;
        st10_is2802m_Result_Data_250_bytes_4_InputAddress_100 AT %IW1731: WORD;
        st10_is2802m_Result_Data_250_bytes_4_InputAddress_101 AT %IW1733: WORD;
        st10_is2802m_Result_Data_250_bytes_4_InputAddress_102 AT %IW1735: WORD;
        st10_is2802m_Result_Data_250_bytes_4_InputAddress_103 AT %IW1737: WORD;
        st10_is2802m_Result_Data_250_bytes_4_InputAddress_104 AT %IW1739: WORD;
        st10_is2802m_Result_Data_250_bytes_4_InputAddress_105 AT %IW1741: WORD;
        st10_is2802m_Result_Data_250_bytes_4_InputAddress_106 AT %IW1743: WORD;
        st10_is2802m_Result_Data_250_bytes_4_InputAddress_107 AT %IW1745: WORD;
        st10_is2802m_Result_Data_250_bytes_4_InputAddress_108 AT %IW1747: WORD;
        st10_is2802m_Result_Data_250_bytes_4_InputAddress_109 AT %IW1749: WORD;
        st10_is2802m_Result_Data_250_bytes_4_InputAddress_110 AT %IW1751: WORD;
        st10_is2802m_Result_Data_250_bytes_4_InputAddress_111 AT %IW1753: WORD;
        st10_is2802m_Result_Data_250_bytes_4_InputAddress_112 AT %IW1755: WORD;
        st10_is2802m_Result_Data_250_bytes_4_InputAddress_113 AT %IW1757: WORD;
        st10_is2802m_Result_Data_250_bytes_4_InputAddress_114 AT %IW1759: WORD;
        st10_is2802m_Result_Data_250_bytes_4_InputAddress_115 AT %IW1761: WORD;
        st10_is2802m_Result_Data_250_bytes_4_InputAddress_116 AT %IW1763: WORD;
        st10_is2802m_Result_Data_250_bytes_4_InputAddress_117 AT %IW1765: WORD;
        st10_is2802m_Result_Data_250_bytes_4_InputAddress_118 AT %IW1767: WORD;
        st10_is2802m_Result_Data_250_bytes_4_InputAddress_119 AT %IW1769: WORD;
        st10_is2802m_Result_Data_250_bytes_4_InputAddress_120 AT %IW1771: WORD;
        st10_is2802m_Result_Data_250_bytes_4_InputAddress_121 AT %IW1773: WORD;
        st10_is2802m_Result_Data_250_bytes_4_InputAddress_122 AT %IW1775: WORD;
        st10_is2802m_Result_Data_250_bytes_4_InputAddress_123 AT %IW1777: WORD;
        st10_is2802m_Result_Data_250_bytes_4_InputAddress_124 AT %IW1779: WORD;
        st10_is2802m_SoftEvent_Control_InputAddress AT %IB2547: BYTE;
        st10_is2802m_SoftEvent_Control_OutputAddress AT %QB2506: BYTE;
        st10_is2802m_User_Data_254_bytes_1_OutputAddress_0 AT %QW2250: WORD;
        st10_is2802m_User_Data_254_bytes_1_OutputAddress_1 AT %QW2252: WORD;
        st10_is2802m_User_Data_254_bytes_1_OutputAddress_2 AT %QW2254: WORD;
        st10_is2802m_User_Data_254_bytes_1_OutputAddress_3 AT %QW2256: WORD;
        st10_is2802m_User_Data_254_bytes_1_OutputAddress_4 AT %QW2258: WORD;
        st10_is2802m_User_Data_254_bytes_1_OutputAddress_5 AT %QW2260: WORD;
        st10_is2802m_User_Data_254_bytes_1_OutputAddress_6 AT %QW2262: WORD;
        st10_is2802m_User_Data_254_bytes_1_OutputAddress_7 AT %QW2264: WORD;
        st10_is2802m_User_Data_254_bytes_1_OutputAddress_8 AT %QW2266: WORD;
        st10_is2802m_User_Data_254_bytes_1_OutputAddress_9 AT %QW2268: WORD;
        st10_is2802m_User_Data_254_bytes_1_OutputAddress_10 AT %QW2270: WORD;
        st10_is2802m_User_Data_254_bytes_1_OutputAddress_11 AT %QW2272: WORD;
        st10_is2802m_User_Data_254_bytes_1_OutputAddress_12 AT %QW2274: WORD;
        st10_is2802m_User_Data_254_bytes_1_OutputAddress_13 AT %QW2276: WORD;
        st10_is2802m_User_Data_254_bytes_1_OutputAddress_14 AT %QW2278: WORD;
        st10_is2802m_User_Data_254_bytes_1_OutputAddress_15 AT %QW2280: WORD;
        st10_is2802m_User_Data_254_bytes_1_OutputAddress_16 AT %QW2282: WORD;
        st10_is2802m_User_Data_254_bytes_1_OutputAddress_17 AT %QW2284: WORD;
        st10_is2802m_User_Data_254_bytes_1_OutputAddress_18 AT %QW2286: WORD;
        st10_is2802m_User_Data_254_bytes_1_OutputAddress_19 AT %QW2288: WORD;
        st10_is2802m_User_Data_254_bytes_1_OutputAddress_20 AT %QW2290: WORD;
        st10_is2802m_User_Data_254_bytes_1_OutputAddress_21 AT %QW2292: WORD;
        st10_is2802m_User_Data_254_bytes_1_OutputAddress_22 AT %QW2294: WORD;
        st10_is2802m_User_Data_254_bytes_1_OutputAddress_23 AT %QW2296: WORD;
        st10_is2802m_User_Data_254_bytes_1_OutputAddress_24 AT %QW2298: WORD;
        st10_is2802m_User_Data_254_bytes_1_OutputAddress_25 AT %QW2300: WORD;
        st10_is2802m_User_Data_254_bytes_1_OutputAddress_26 AT %QW2302: WORD;
        st10_is2802m_User_Data_254_bytes_1_OutputAddress_27 AT %QW2304: WORD;
        st10_is2802m_User_Data_254_bytes_1_OutputAddress_28 AT %QW2306: WORD;
        st10_is2802m_User_Data_254_bytes_1_OutputAddress_29 AT %QW2308: WORD;
        st10_is2802m_User_Data_254_bytes_1_OutputAddress_30 AT %QW2310: WORD;
        st10_is2802m_User_Data_254_bytes_1_OutputAddress_31 AT %QW2312: WORD;
        st10_is2802m_User_Data_254_bytes_1_OutputAddress_32 AT %QW2314: WORD;
        st10_is2802m_User_Data_254_bytes_1_OutputAddress_33 AT %QW2316: WORD;
        st10_is2802m_User_Data_254_bytes_1_OutputAddress_34 AT %QW2318: WORD;
        st10_is2802m_User_Data_254_bytes_1_OutputAddress_35 AT %QW2320: WORD;
        st10_is2802m_User_Data_254_bytes_1_OutputAddress_36 AT %QW2322: WORD;
        st10_is2802m_User_Data_254_bytes_1_OutputAddress_37 AT %QW2324: WORD;
        st10_is2802m_User_Data_254_bytes_1_OutputAddress_38 AT %QW2326: WORD;
        st10_is2802m_User_Data_254_bytes_1_OutputAddress_39 AT %QW2328: WORD;
        st10_is2802m_User_Data_254_bytes_1_OutputAddress_40 AT %QW2330: WORD;
        st10_is2802m_User_Data_254_bytes_1_OutputAddress_41 AT %QW2332: WORD;
        st10_is2802m_User_Data_254_bytes_1_OutputAddress_42 AT %QW2334: WORD;
        st10_is2802m_User_Data_254_bytes_1_OutputAddress_43 AT %QW2336: WORD;
        st10_is2802m_User_Data_254_bytes_1_OutputAddress_44 AT %QW2338: WORD;
        st10_is2802m_User_Data_254_bytes_1_OutputAddress_45 AT %QW2340: WORD;
        st10_is2802m_User_Data_254_bytes_1_OutputAddress_46 AT %QW2342: WORD;
        st10_is2802m_User_Data_254_bytes_1_OutputAddress_47 AT %QW2344: WORD;
        st10_is2802m_User_Data_254_bytes_1_OutputAddress_48 AT %QW2346: WORD;
        st10_is2802m_User_Data_254_bytes_1_OutputAddress_49 AT %QW2348: WORD;
        st10_is2802m_User_Data_254_bytes_1_OutputAddress_50 AT %QW2350: WORD;
        st10_is2802m_User_Data_254_bytes_1_OutputAddress_51 AT %QW2352: WORD;
        st10_is2802m_User_Data_254_bytes_1_OutputAddress_52 AT %QW2354: WORD;
        st10_is2802m_User_Data_254_bytes_1_OutputAddress_53 AT %QW2356: WORD;
        st10_is2802m_User_Data_254_bytes_1_OutputAddress_54 AT %QW2358: WORD;
        st10_is2802m_User_Data_254_bytes_1_OutputAddress_55 AT %QW2360: WORD;
        st10_is2802m_User_Data_254_bytes_1_OutputAddress_56 AT %QW2362: WORD;
        st10_is2802m_User_Data_254_bytes_1_OutputAddress_57 AT %QW2364: WORD;
        st10_is2802m_User_Data_254_bytes_1_OutputAddress_58 AT %QW2366: WORD;
        st10_is2802m_User_Data_254_bytes_1_OutputAddress_59 AT %QW2368: WORD;
        st10_is2802m_User_Data_254_bytes_1_OutputAddress_60 AT %QW2370: WORD;
        st10_is2802m_User_Data_254_bytes_1_OutputAddress_61 AT %QW2372: WORD;
        st10_is2802m_User_Data_254_bytes_1_OutputAddress_62 AT %QW2374: WORD;
        st10_is2802m_User_Data_254_bytes_1_OutputAddress_63 AT %QW2376: WORD;
        st10_is2802m_User_Data_254_bytes_1_OutputAddress_64 AT %QW2378: WORD;
        st10_is2802m_User_Data_254_bytes_1_OutputAddress_65 AT %QW2380: WORD;
        st10_is2802m_User_Data_254_bytes_1_OutputAddress_66 AT %QW2382: WORD;
        st10_is2802m_User_Data_254_bytes_1_OutputAddress_67 AT %QW2384: WORD;
        st10_is2802m_User_Data_254_bytes_1_OutputAddress_68 AT %QW2386: WORD;
        st10_is2802m_User_Data_254_bytes_1_OutputAddress_69 AT %QW2388: WORD;
        st10_is2802m_User_Data_254_bytes_1_OutputAddress_70 AT %QW2390: WORD;
        st10_is2802m_User_Data_254_bytes_1_OutputAddress_71 AT %QW2392: WORD;
        st10_is2802m_User_Data_254_bytes_1_OutputAddress_72 AT %QW2394: WORD;
        st10_is2802m_User_Data_254_bytes_1_OutputAddress_73 AT %QW2396: WORD;
        st10_is2802m_User_Data_254_bytes_1_OutputAddress_74 AT %QW2398: WORD;
        st10_is2802m_User_Data_254_bytes_1_OutputAddress_75 AT %QW2400: WORD;
        st10_is2802m_User_Data_254_bytes_1_OutputAddress_76 AT %QW2402: WORD;
        st10_is2802m_User_Data_254_bytes_1_OutputAddress_77 AT %QW2404: WORD;
        st10_is2802m_User_Data_254_bytes_1_OutputAddress_78 AT %QW2406: WORD;
        st10_is2802m_User_Data_254_bytes_1_OutputAddress_79 AT %QW2408: WORD;
        st10_is2802m_User_Data_254_bytes_1_OutputAddress_80 AT %QW2410: WORD;
        st10_is2802m_User_Data_254_bytes_1_OutputAddress_81 AT %QW2412: WORD;
        st10_is2802m_User_Data_254_bytes_1_OutputAddress_82 AT %QW2414: WORD;
        st10_is2802m_User_Data_254_bytes_1_OutputAddress_83 AT %QW2416: WORD;
        st10_is2802m_User_Data_254_bytes_1_OutputAddress_84 AT %QW2418: WORD;
        st10_is2802m_User_Data_254_bytes_1_OutputAddress_85 AT %QW2420: WORD;
        st10_is2802m_User_Data_254_bytes_1_OutputAddress_86 AT %QW2422: WORD;
        st10_is2802m_User_Data_254_bytes_1_OutputAddress_87 AT %QW2424: WORD;
        st10_is2802m_User_Data_254_bytes_1_OutputAddress_88 AT %QW2426: WORD;
        st10_is2802m_User_Data_254_bytes_1_OutputAddress_89 AT %QW2428: WORD;
        st10_is2802m_User_Data_254_bytes_1_OutputAddress_90 AT %QW2430: WORD;
        st10_is2802m_User_Data_254_bytes_1_OutputAddress_91 AT %QW2432: WORD;
        st10_is2802m_User_Data_254_bytes_1_OutputAddress_92 AT %QW2434: WORD;
        st10_is2802m_User_Data_254_bytes_1_OutputAddress_93 AT %QW2436: WORD;
        st10_is2802m_User_Data_254_bytes_1_OutputAddress_94 AT %QW2438: WORD;
        st10_is2802m_User_Data_254_bytes_1_OutputAddress_95 AT %QW2440: WORD;
        st10_is2802m_User_Data_254_bytes_1_OutputAddress_96 AT %QW2442: WORD;
        st10_is2802m_User_Data_254_bytes_1_OutputAddress_97 AT %QW2444: WORD;
        st10_is2802m_User_Data_254_bytes_1_OutputAddress_98 AT %QW2446: WORD;
        st10_is2802m_User_Data_254_bytes_1_OutputAddress_99 AT %QW2448: WORD;
        st10_is2802m_User_Data_254_bytes_1_OutputAddress_100 AT %QW2450: WORD;
        st10_is2802m_User_Data_254_bytes_1_OutputAddress_101 AT %QW2452: WORD;
        st10_is2802m_User_Data_254_bytes_1_OutputAddress_102 AT %QW2454: WORD;
        st10_is2802m_User_Data_254_bytes_1_OutputAddress_103 AT %QW2456: WORD;
        st10_is2802m_User_Data_254_bytes_1_OutputAddress_104 AT %QW2458: WORD;
        st10_is2802m_User_Data_254_bytes_1_OutputAddress_105 AT %QW2460: WORD;
        st10_is2802m_User_Data_254_bytes_1_OutputAddress_106 AT %QW2462: WORD;
        st10_is2802m_User_Data_254_bytes_1_OutputAddress_107 AT %QW2464: WORD;
        st10_is2802m_User_Data_254_bytes_1_OutputAddress_108 AT %QW2466: WORD;
        st10_is2802m_User_Data_254_bytes_1_OutputAddress_109 AT %QW2468: WORD;
        st10_is2802m_User_Data_254_bytes_1_OutputAddress_110 AT %QW2470: WORD;
        st10_is2802m_User_Data_254_bytes_1_OutputAddress_111 AT %QW2472: WORD;
        st10_is2802m_User_Data_254_bytes_1_OutputAddress_112 AT %QW2474: WORD;
        st10_is2802m_User_Data_254_bytes_1_OutputAddress_113 AT %QW2476: WORD;
        st10_is2802m_User_Data_254_bytes_1_OutputAddress_114 AT %QW2478: WORD;
        st10_is2802m_User_Data_254_bytes_1_OutputAddress_115 AT %QW2480: WORD;
        st10_is2802m_User_Data_254_bytes_1_OutputAddress_116 AT %QW2482: WORD;
        st10_is2802m_User_Data_254_bytes_1_OutputAddress_117 AT %QW2484: WORD;
        st10_is2802m_User_Data_254_bytes_1_OutputAddress_118 AT %QW2486: WORD;
        st10_is2802m_User_Data_254_bytes_1_OutputAddress_119 AT %QW2488: WORD;
        st10_is2802m_User_Data_254_bytes_1_OutputAddress_120 AT %QW2490: WORD;
        st10_is2802m_User_Data_254_bytes_1_OutputAddress_121 AT %QW2492: WORD;
        st10_is2802m_User_Data_254_bytes_1_OutputAddress_122 AT %QW2494: WORD;
        st10_is2802m_User_Data_254_bytes_1_OutputAddress_123 AT %QW2496: WORD;
        st10_is2802m_User_Data_254_bytes_1_OutputAddress_124 AT %QW2498: WORD;
        st10_is2802m_User_Data_254_bytes_1_OutputAddress_125 AT %QW2500: WORD;
        st10_is2802m_User_Data_254_bytes_1_OutputAddress_126 AT %QW2502: WORD;
        st10_is2802m_User_Data_254_bytes_2_OutputAddress_0 AT %QW1996: WORD;
        st10_is2802m_User_Data_254_bytes_2_OutputAddress_1 AT %QW1998: WORD;
        st10_is2802m_User_Data_254_bytes_2_OutputAddress_2 AT %QW2000: WORD;
        st10_is2802m_User_Data_254_bytes_2_OutputAddress_3 AT %QW2002: WORD;
        st10_is2802m_User_Data_254_bytes_2_OutputAddress_4 AT %QW2004: WORD;
        st10_is2802m_User_Data_254_bytes_2_OutputAddress_5 AT %QW2006: WORD;
        st10_is2802m_User_Data_254_bytes_2_OutputAddress_6 AT %QW2008: WORD;
        st10_is2802m_User_Data_254_bytes_2_OutputAddress_7 AT %QW2010: WORD;
        st10_is2802m_User_Data_254_bytes_2_OutputAddress_8 AT %QW2012: WORD;
        st10_is2802m_User_Data_254_bytes_2_OutputAddress_9 AT %QW2014: WORD;
        st10_is2802m_User_Data_254_bytes_2_OutputAddress_10 AT %QW2016: WORD;
        st10_is2802m_User_Data_254_bytes_2_OutputAddress_11 AT %QW2018: WORD;
        st10_is2802m_User_Data_254_bytes_2_OutputAddress_12 AT %QW2020: WORD;
        st10_is2802m_User_Data_254_bytes_2_OutputAddress_13 AT %QW2022: WORD;
        st10_is2802m_User_Data_254_bytes_2_OutputAddress_14 AT %QW2024: WORD;
        st10_is2802m_User_Data_254_bytes_2_OutputAddress_15 AT %QW2026: WORD;
        st10_is2802m_User_Data_254_bytes_2_OutputAddress_16 AT %QW2028: WORD;
        st10_is2802m_User_Data_254_bytes_2_OutputAddress_17 AT %QW2030: WORD;
        st10_is2802m_User_Data_254_bytes_2_OutputAddress_18 AT %QW2032: WORD;
        st10_is2802m_User_Data_254_bytes_2_OutputAddress_19 AT %QW2034: WORD;
        st10_is2802m_User_Data_254_bytes_2_OutputAddress_20 AT %QW2036: WORD;
        st10_is2802m_User_Data_254_bytes_2_OutputAddress_21 AT %QW2038: WORD;
        st10_is2802m_User_Data_254_bytes_2_OutputAddress_22 AT %QW2040: WORD;
        st10_is2802m_User_Data_254_bytes_2_OutputAddress_23 AT %QW2042: WORD;
        st10_is2802m_User_Data_254_bytes_2_OutputAddress_24 AT %QW2044: WORD;
        st10_is2802m_User_Data_254_bytes_2_OutputAddress_25 AT %QW2046: WORD;
        st10_is2802m_User_Data_254_bytes_2_OutputAddress_26 AT %QW2048: WORD;
        st10_is2802m_User_Data_254_bytes_2_OutputAddress_27 AT %QW2050: WORD;
        st10_is2802m_User_Data_254_bytes_2_OutputAddress_28 AT %QW2052: WORD;
        st10_is2802m_User_Data_254_bytes_2_OutputAddress_29 AT %QW2054: WORD;
        st10_is2802m_User_Data_254_bytes_2_OutputAddress_30 AT %QW2056: WORD;
        st10_is2802m_User_Data_254_bytes_2_OutputAddress_31 AT %QW2058: WORD;
        st10_is2802m_User_Data_254_bytes_2_OutputAddress_32 AT %QW2060: WORD;
        st10_is2802m_User_Data_254_bytes_2_OutputAddress_33 AT %QW2062: WORD;
        st10_is2802m_User_Data_254_bytes_2_OutputAddress_34 AT %QW2064: WORD;
        st10_is2802m_User_Data_254_bytes_2_OutputAddress_35 AT %QW2066: WORD;
        st10_is2802m_User_Data_254_bytes_2_OutputAddress_36 AT %QW2068: WORD;
        st10_is2802m_User_Data_254_bytes_2_OutputAddress_37 AT %QW2070: WORD;
        st10_is2802m_User_Data_254_bytes_2_OutputAddress_38 AT %QW2072: WORD;
        st10_is2802m_User_Data_254_bytes_2_OutputAddress_39 AT %QW2074: WORD;
        st10_is2802m_User_Data_254_bytes_2_OutputAddress_40 AT %QW2076: WORD;
        st10_is2802m_User_Data_254_bytes_2_OutputAddress_41 AT %QW2078: WORD;
        st10_is2802m_User_Data_254_bytes_2_OutputAddress_42 AT %QW2080: WORD;
        st10_is2802m_User_Data_254_bytes_2_OutputAddress_43 AT %QW2082: WORD;
        st10_is2802m_User_Data_254_bytes_2_OutputAddress_44 AT %QW2084: WORD;
        st10_is2802m_User_Data_254_bytes_2_OutputAddress_45 AT %QW2086: WORD;
        st10_is2802m_User_Data_254_bytes_2_OutputAddress_46 AT %QW2088: WORD;
        st10_is2802m_User_Data_254_bytes_2_OutputAddress_47 AT %QW2090: WORD;
        st10_is2802m_User_Data_254_bytes_2_OutputAddress_48 AT %QW2092: WORD;
        st10_is2802m_User_Data_254_bytes_2_OutputAddress_49 AT %QW2094: WORD;
        st10_is2802m_User_Data_254_bytes_2_OutputAddress_50 AT %QW2096: WORD;
        st10_is2802m_User_Data_254_bytes_2_OutputAddress_51 AT %QW2098: WORD;
        st10_is2802m_User_Data_254_bytes_2_OutputAddress_52 AT %QW2100: WORD;
        st10_is2802m_User_Data_254_bytes_2_OutputAddress_53 AT %QW2102: WORD;
        st10_is2802m_User_Data_254_bytes_2_OutputAddress_54 AT %QW2104: WORD;
        st10_is2802m_User_Data_254_bytes_2_OutputAddress_55 AT %QW2106: WORD;
        st10_is2802m_User_Data_254_bytes_2_OutputAddress_56 AT %QW2108: WORD;
        st10_is2802m_User_Data_254_bytes_2_OutputAddress_57 AT %QW2110: WORD;
        st10_is2802m_User_Data_254_bytes_2_OutputAddress_58 AT %QW2112: WORD;
        st10_is2802m_User_Data_254_bytes_2_OutputAddress_59 AT %QW2114: WORD;
        st10_is2802m_User_Data_254_bytes_2_OutputAddress_60 AT %QW2116: WORD;
        st10_is2802m_User_Data_254_bytes_2_OutputAddress_61 AT %QW2118: WORD;
        st10_is2802m_User_Data_254_bytes_2_OutputAddress_62 AT %QW2120: WORD;
        st10_is2802m_User_Data_254_bytes_2_OutputAddress_63 AT %QW2122: WORD;
        st10_is2802m_User_Data_254_bytes_2_OutputAddress_64 AT %QW2124: WORD;
        st10_is2802m_User_Data_254_bytes_2_OutputAddress_65 AT %QW2126: WORD;
        st10_is2802m_User_Data_254_bytes_2_OutputAddress_66 AT %QW2128: WORD;
        st10_is2802m_User_Data_254_bytes_2_OutputAddress_67 AT %QW2130: WORD;
        st10_is2802m_User_Data_254_bytes_2_OutputAddress_68 AT %QW2132: WORD;
        st10_is2802m_User_Data_254_bytes_2_OutputAddress_69 AT %QW2134: WORD;
        st10_is2802m_User_Data_254_bytes_2_OutputAddress_70 AT %QW2136: WORD;
        st10_is2802m_User_Data_254_bytes_2_OutputAddress_71 AT %QW2138: WORD;
        st10_is2802m_User_Data_254_bytes_2_OutputAddress_72 AT %QW2140: WORD;
        st10_is2802m_User_Data_254_bytes_2_OutputAddress_73 AT %QW2142: WORD;
        st10_is2802m_User_Data_254_bytes_2_OutputAddress_74 AT %QW2144: WORD;
        st10_is2802m_User_Data_254_bytes_2_OutputAddress_75 AT %QW2146: WORD;
        st10_is2802m_User_Data_254_bytes_2_OutputAddress_76 AT %QW2148: WORD;
        st10_is2802m_User_Data_254_bytes_2_OutputAddress_77 AT %QW2150: WORD;
        st10_is2802m_User_Data_254_bytes_2_OutputAddress_78 AT %QW2152: WORD;
        st10_is2802m_User_Data_254_bytes_2_OutputAddress_79 AT %QW2154: WORD;
        st10_is2802m_User_Data_254_bytes_2_OutputAddress_80 AT %QW2156: WORD;
        st10_is2802m_User_Data_254_bytes_2_OutputAddress_81 AT %QW2158: WORD;
        st10_is2802m_User_Data_254_bytes_2_OutputAddress_82 AT %QW2160: WORD;
        st10_is2802m_User_Data_254_bytes_2_OutputAddress_83 AT %QW2162: WORD;
        st10_is2802m_User_Data_254_bytes_2_OutputAddress_84 AT %QW2164: WORD;
        st10_is2802m_User_Data_254_bytes_2_OutputAddress_85 AT %QW2166: WORD;
        st10_is2802m_User_Data_254_bytes_2_OutputAddress_86 AT %QW2168: WORD;
        st10_is2802m_User_Data_254_bytes_2_OutputAddress_87 AT %QW2170: WORD;
        st10_is2802m_User_Data_254_bytes_2_OutputAddress_88 AT %QW2172: WORD;
        st10_is2802m_User_Data_254_bytes_2_OutputAddress_89 AT %QW2174: WORD;
        st10_is2802m_User_Data_254_bytes_2_OutputAddress_90 AT %QW2176: WORD;
        st10_is2802m_User_Data_254_bytes_2_OutputAddress_91 AT %QW2178: WORD;
        st10_is2802m_User_Data_254_bytes_2_OutputAddress_92 AT %QW2180: WORD;
        st10_is2802m_User_Data_254_bytes_2_OutputAddress_93 AT %QW2182: WORD;
        st10_is2802m_User_Data_254_bytes_2_OutputAddress_94 AT %QW2184: WORD;
        st10_is2802m_User_Data_254_bytes_2_OutputAddress_95 AT %QW2186: WORD;
        st10_is2802m_User_Data_254_bytes_2_OutputAddress_96 AT %QW2188: WORD;
        st10_is2802m_User_Data_254_bytes_2_OutputAddress_97 AT %QW2190: WORD;
        st10_is2802m_User_Data_254_bytes_2_OutputAddress_98 AT %QW2192: WORD;
        st10_is2802m_User_Data_254_bytes_2_OutputAddress_99 AT %QW2194: WORD;
        st10_is2802m_User_Data_254_bytes_2_OutputAddress_100 AT %QW2196: WORD;
        st10_is2802m_User_Data_254_bytes_2_OutputAddress_101 AT %QW2198: WORD;
        st10_is2802m_User_Data_254_bytes_2_OutputAddress_102 AT %QW2200: WORD;
        st10_is2802m_User_Data_254_bytes_2_OutputAddress_103 AT %QW2202: WORD;
        st10_is2802m_User_Data_254_bytes_2_OutputAddress_104 AT %QW2204: WORD;
        st10_is2802m_User_Data_254_bytes_2_OutputAddress_105 AT %QW2206: WORD;
        st10_is2802m_User_Data_254_bytes_2_OutputAddress_106 AT %QW2208: WORD;
        st10_is2802m_User_Data_254_bytes_2_OutputAddress_107 AT %QW2210: WORD;
        st10_is2802m_User_Data_254_bytes_2_OutputAddress_108 AT %QW2212: WORD;
        st10_is2802m_User_Data_254_bytes_2_OutputAddress_109 AT %QW2214: WORD;
        st10_is2802m_User_Data_254_bytes_2_OutputAddress_110 AT %QW2216: WORD;
        st10_is2802m_User_Data_254_bytes_2_OutputAddress_111 AT %QW2218: WORD;
        st10_is2802m_User_Data_254_bytes_2_OutputAddress_112 AT %QW2220: WORD;
        st10_is2802m_User_Data_254_bytes_2_OutputAddress_113 AT %QW2222: WORD;
        st10_is2802m_User_Data_254_bytes_2_OutputAddress_114 AT %QW2224: WORD;
        st10_is2802m_User_Data_254_bytes_2_OutputAddress_115 AT %QW2226: WORD;
        st10_is2802m_User_Data_254_bytes_2_OutputAddress_116 AT %QW2228: WORD;
        st10_is2802m_User_Data_254_bytes_2_OutputAddress_117 AT %QW2230: WORD;
        st10_is2802m_User_Data_254_bytes_2_OutputAddress_118 AT %QW2232: WORD;
        st10_is2802m_User_Data_254_bytes_2_OutputAddress_119 AT %QW2234: WORD;
        st10_is2802m_User_Data_254_bytes_2_OutputAddress_120 AT %QW2236: WORD;
        st10_is2802m_User_Data_254_bytes_2_OutputAddress_121 AT %QW2238: WORD;
        st10_is2802m_User_Data_254_bytes_2_OutputAddress_122 AT %QW2240: WORD;
        st10_is2802m_User_Data_254_bytes_2_OutputAddress_123 AT %QW2242: WORD;
        st10_is2802m_User_Data_254_bytes_2_OutputAddress_124 AT %QW2244: WORD;
        st10_is2802m_User_Data_254_bytes_2_OutputAddress_125 AT %QW2246: WORD;
        st10_is2802m_User_Data_254_bytes_2_OutputAddress_126 AT %QW2248: WORD;
        st10_is2802m_User_Data_254_bytes_3_OutputAddress_0 AT %QW1742: WORD;
        st10_is2802m_User_Data_254_bytes_3_OutputAddress_1 AT %QW1744: WORD;
        st10_is2802m_User_Data_254_bytes_3_OutputAddress_2 AT %QW1746: WORD;
        st10_is2802m_User_Data_254_bytes_3_OutputAddress_3 AT %QW1748: WORD;
        st10_is2802m_User_Data_254_bytes_3_OutputAddress_4 AT %QW1750: WORD;
        st10_is2802m_User_Data_254_bytes_3_OutputAddress_5 AT %QW1752: WORD;
        st10_is2802m_User_Data_254_bytes_3_OutputAddress_6 AT %QW1754: WORD;
        st10_is2802m_User_Data_254_bytes_3_OutputAddress_7 AT %QW1756: WORD;
        st10_is2802m_User_Data_254_bytes_3_OutputAddress_8 AT %QW1758: WORD;
        st10_is2802m_User_Data_254_bytes_3_OutputAddress_9 AT %QW1760: WORD;
        st10_is2802m_User_Data_254_bytes_3_OutputAddress_10 AT %QW1762: WORD;
        st10_is2802m_User_Data_254_bytes_3_OutputAddress_11 AT %QW1764: WORD;
        st10_is2802m_User_Data_254_bytes_3_OutputAddress_12 AT %QW1766: WORD;
        st10_is2802m_User_Data_254_bytes_3_OutputAddress_13 AT %QW1768: WORD;
        st10_is2802m_User_Data_254_bytes_3_OutputAddress_14 AT %QW1770: WORD;
        st10_is2802m_User_Data_254_bytes_3_OutputAddress_15 AT %QW1772: WORD;
        st10_is2802m_User_Data_254_bytes_3_OutputAddress_16 AT %QW1774: WORD;
        st10_is2802m_User_Data_254_bytes_3_OutputAddress_17 AT %QW1776: WORD;
        st10_is2802m_User_Data_254_bytes_3_OutputAddress_18 AT %QW1778: WORD;
        st10_is2802m_User_Data_254_bytes_3_OutputAddress_19 AT %QW1780: WORD;
        st10_is2802m_User_Data_254_bytes_3_OutputAddress_20 AT %QW1782: WORD;
        st10_is2802m_User_Data_254_bytes_3_OutputAddress_21 AT %QW1784: WORD;
        st10_is2802m_User_Data_254_bytes_3_OutputAddress_22 AT %QW1786: WORD;
        st10_is2802m_User_Data_254_bytes_3_OutputAddress_23 AT %QW1788: WORD;
        st10_is2802m_User_Data_254_bytes_3_OutputAddress_24 AT %QW1790: WORD;
        st10_is2802m_User_Data_254_bytes_3_OutputAddress_25 AT %QW1792: WORD;
        st10_is2802m_User_Data_254_bytes_3_OutputAddress_26 AT %QW1794: WORD;
        st10_is2802m_User_Data_254_bytes_3_OutputAddress_27 AT %QW1796: WORD;
        st10_is2802m_User_Data_254_bytes_3_OutputAddress_28 AT %QW1798: WORD;
        st10_is2802m_User_Data_254_bytes_3_OutputAddress_29 AT %QW1800: WORD;
        st10_is2802m_User_Data_254_bytes_3_OutputAddress_30 AT %QW1802: WORD;
        st10_is2802m_User_Data_254_bytes_3_OutputAddress_31 AT %QW1804: WORD;
        st10_is2802m_User_Data_254_bytes_3_OutputAddress_32 AT %QW1806: WORD;
        st10_is2802m_User_Data_254_bytes_3_OutputAddress_33 AT %QW1808: WORD;
        st10_is2802m_User_Data_254_bytes_3_OutputAddress_34 AT %QW1810: WORD;
        st10_is2802m_User_Data_254_bytes_3_OutputAddress_35 AT %QW1812: WORD;
        st10_is2802m_User_Data_254_bytes_3_OutputAddress_36 AT %QW1814: WORD;
        st10_is2802m_User_Data_254_bytes_3_OutputAddress_37 AT %QW1816: WORD;
        st10_is2802m_User_Data_254_bytes_3_OutputAddress_38 AT %QW1818: WORD;
        st10_is2802m_User_Data_254_bytes_3_OutputAddress_39 AT %QW1820: WORD;
        st10_is2802m_User_Data_254_bytes_3_OutputAddress_40 AT %QW1822: WORD;
        st10_is2802m_User_Data_254_bytes_3_OutputAddress_41 AT %QW1824: WORD;
        st10_is2802m_User_Data_254_bytes_3_OutputAddress_42 AT %QW1826: WORD;
        st10_is2802m_User_Data_254_bytes_3_OutputAddress_43 AT %QW1828: WORD;
        st10_is2802m_User_Data_254_bytes_3_OutputAddress_44 AT %QW1830: WORD;
        st10_is2802m_User_Data_254_bytes_3_OutputAddress_45 AT %QW1832: WORD;
        st10_is2802m_User_Data_254_bytes_3_OutputAddress_46 AT %QW1834: WORD;
        st10_is2802m_User_Data_254_bytes_3_OutputAddress_47 AT %QW1836: WORD;
        st10_is2802m_User_Data_254_bytes_3_OutputAddress_48 AT %QW1838: WORD;
        st10_is2802m_User_Data_254_bytes_3_OutputAddress_49 AT %QW1840: WORD;
        st10_is2802m_User_Data_254_bytes_3_OutputAddress_50 AT %QW1842: WORD;
        st10_is2802m_User_Data_254_bytes_3_OutputAddress_51 AT %QW1844: WORD;
        st10_is2802m_User_Data_254_bytes_3_OutputAddress_52 AT %QW1846: WORD;
        st10_is2802m_User_Data_254_bytes_3_OutputAddress_53 AT %QW1848: WORD;
        st10_is2802m_User_Data_254_bytes_3_OutputAddress_54 AT %QW1850: WORD;
        st10_is2802m_User_Data_254_bytes_3_OutputAddress_55 AT %QW1852: WORD;
        st10_is2802m_User_Data_254_bytes_3_OutputAddress_56 AT %QW1854: WORD;
        st10_is2802m_User_Data_254_bytes_3_OutputAddress_57 AT %QW1856: WORD;
        st10_is2802m_User_Data_254_bytes_3_OutputAddress_58 AT %QW1858: WORD;
        st10_is2802m_User_Data_254_bytes_3_OutputAddress_59 AT %QW1860: WORD;
        st10_is2802m_User_Data_254_bytes_3_OutputAddress_60 AT %QW1862: WORD;
        st10_is2802m_User_Data_254_bytes_3_OutputAddress_61 AT %QW1864: WORD;
        st10_is2802m_User_Data_254_bytes_3_OutputAddress_62 AT %QW1866: WORD;
        st10_is2802m_User_Data_254_bytes_3_OutputAddress_63 AT %QW1868: WORD;
        st10_is2802m_User_Data_254_bytes_3_OutputAddress_64 AT %QW1870: WORD;
        st10_is2802m_User_Data_254_bytes_3_OutputAddress_65 AT %QW1872: WORD;
        st10_is2802m_User_Data_254_bytes_3_OutputAddress_66 AT %QW1874: WORD;
        st10_is2802m_User_Data_254_bytes_3_OutputAddress_67 AT %QW1876: WORD;
        st10_is2802m_User_Data_254_bytes_3_OutputAddress_68 AT %QW1878: WORD;
        st10_is2802m_User_Data_254_bytes_3_OutputAddress_69 AT %QW1880: WORD;
        st10_is2802m_User_Data_254_bytes_3_OutputAddress_70 AT %QW1882: WORD;
        st10_is2802m_User_Data_254_bytes_3_OutputAddress_71 AT %QW1884: WORD;
        st10_is2802m_User_Data_254_bytes_3_OutputAddress_72 AT %QW1886: WORD;
        st10_is2802m_User_Data_254_bytes_3_OutputAddress_73 AT %QW1888: WORD;
        st10_is2802m_User_Data_254_bytes_3_OutputAddress_74 AT %QW1890: WORD;
        st10_is2802m_User_Data_254_bytes_3_OutputAddress_75 AT %QW1892: WORD;
        st10_is2802m_User_Data_254_bytes_3_OutputAddress_76 AT %QW1894: WORD;
        st10_is2802m_User_Data_254_bytes_3_OutputAddress_77 AT %QW1896: WORD;
        st10_is2802m_User_Data_254_bytes_3_OutputAddress_78 AT %QW1898: WORD;
        st10_is2802m_User_Data_254_bytes_3_OutputAddress_79 AT %QW1900: WORD;
        st10_is2802m_User_Data_254_bytes_3_OutputAddress_80 AT %QW1902: WORD;
        st10_is2802m_User_Data_254_bytes_3_OutputAddress_81 AT %QW1904: WORD;
        st10_is2802m_User_Data_254_bytes_3_OutputAddress_82 AT %QW1906: WORD;
        st10_is2802m_User_Data_254_bytes_3_OutputAddress_83 AT %QW1908: WORD;
        st10_is2802m_User_Data_254_bytes_3_OutputAddress_84 AT %QW1910: WORD;
        st10_is2802m_User_Data_254_bytes_3_OutputAddress_85 AT %QW1912: WORD;
        st10_is2802m_User_Data_254_bytes_3_OutputAddress_86 AT %QW1914: WORD;
        st10_is2802m_User_Data_254_bytes_3_OutputAddress_87 AT %QW1916: WORD;
        st10_is2802m_User_Data_254_bytes_3_OutputAddress_88 AT %QW1918: WORD;
        st10_is2802m_User_Data_254_bytes_3_OutputAddress_89 AT %QW1920: WORD;
        st10_is2802m_User_Data_254_bytes_3_OutputAddress_90 AT %QW1922: WORD;
        st10_is2802m_User_Data_254_bytes_3_OutputAddress_91 AT %QW1924: WORD;
        st10_is2802m_User_Data_254_bytes_3_OutputAddress_92 AT %QW1926: WORD;
        st10_is2802m_User_Data_254_bytes_3_OutputAddress_93 AT %QW1928: WORD;
        st10_is2802m_User_Data_254_bytes_3_OutputAddress_94 AT %QW1930: WORD;
        st10_is2802m_User_Data_254_bytes_3_OutputAddress_95 AT %QW1932: WORD;
        st10_is2802m_User_Data_254_bytes_3_OutputAddress_96 AT %QW1934: WORD;
        st10_is2802m_User_Data_254_bytes_3_OutputAddress_97 AT %QW1936: WORD;
        st10_is2802m_User_Data_254_bytes_3_OutputAddress_98 AT %QW1938: WORD;
        st10_is2802m_User_Data_254_bytes_3_OutputAddress_99 AT %QW1940: WORD;
        st10_is2802m_User_Data_254_bytes_3_OutputAddress_100 AT %QW1942: WORD;
        st10_is2802m_User_Data_254_bytes_3_OutputAddress_101 AT %QW1944: WORD;
        st10_is2802m_User_Data_254_bytes_3_OutputAddress_102 AT %QW1946: WORD;
        st10_is2802m_User_Data_254_bytes_3_OutputAddress_103 AT %QW1948: WORD;
        st10_is2802m_User_Data_254_bytes_3_OutputAddress_104 AT %QW1950: WORD;
        st10_is2802m_User_Data_254_bytes_3_OutputAddress_105 AT %QW1952: WORD;
        st10_is2802m_User_Data_254_bytes_3_OutputAddress_106 AT %QW1954: WORD;
        st10_is2802m_User_Data_254_bytes_3_OutputAddress_107 AT %QW1956: WORD;
        st10_is2802m_User_Data_254_bytes_3_OutputAddress_108 AT %QW1958: WORD;
        st10_is2802m_User_Data_254_bytes_3_OutputAddress_109 AT %QW1960: WORD;
        st10_is2802m_User_Data_254_bytes_3_OutputAddress_110 AT %QW1962: WORD;
        st10_is2802m_User_Data_254_bytes_3_OutputAddress_111 AT %QW1964: WORD;
        st10_is2802m_User_Data_254_bytes_3_OutputAddress_112 AT %QW1966: WORD;
        st10_is2802m_User_Data_254_bytes_3_OutputAddress_113 AT %QW1968: WORD;
        st10_is2802m_User_Data_254_bytes_3_OutputAddress_114 AT %QW1970: WORD;
        st10_is2802m_User_Data_254_bytes_3_OutputAddress_115 AT %QW1972: WORD;
        st10_is2802m_User_Data_254_bytes_3_OutputAddress_116 AT %QW1974: WORD;
        st10_is2802m_User_Data_254_bytes_3_OutputAddress_117 AT %QW1976: WORD;
        st10_is2802m_User_Data_254_bytes_3_OutputAddress_118 AT %QW1978: WORD;
        st10_is2802m_User_Data_254_bytes_3_OutputAddress_119 AT %QW1980: WORD;
        st10_is2802m_User_Data_254_bytes_3_OutputAddress_120 AT %QW1982: WORD;
        st10_is2802m_User_Data_254_bytes_3_OutputAddress_121 AT %QW1984: WORD;
        st10_is2802m_User_Data_254_bytes_3_OutputAddress_122 AT %QW1986: WORD;
        st10_is2802m_User_Data_254_bytes_3_OutputAddress_123 AT %QW1988: WORD;
        st10_is2802m_User_Data_254_bytes_3_OutputAddress_124 AT %QW1990: WORD;
        st10_is2802m_User_Data_254_bytes_3_OutputAddress_125 AT %QW1992: WORD;
        st10_is2802m_User_Data_254_bytes_3_OutputAddress_126 AT %QW1994: WORD;
        st10_is2802m_User_Data_254_bytes_4_OutputAddress_0 AT %QW1488: WORD;
        st10_is2802m_User_Data_254_bytes_4_OutputAddress_1 AT %QW1490: WORD;
        st10_is2802m_User_Data_254_bytes_4_OutputAddress_2 AT %QW1492: WORD;
        st10_is2802m_User_Data_254_bytes_4_OutputAddress_3 AT %QW1494: WORD;
        st10_is2802m_User_Data_254_bytes_4_OutputAddress_4 AT %QW1496: WORD;
        st10_is2802m_User_Data_254_bytes_4_OutputAddress_5 AT %QW1498: WORD;
        st10_is2802m_User_Data_254_bytes_4_OutputAddress_6 AT %QW1500: WORD;
        st10_is2802m_User_Data_254_bytes_4_OutputAddress_7 AT %QW1502: WORD;
        st10_is2802m_User_Data_254_bytes_4_OutputAddress_8 AT %QW1504: WORD;
        st10_is2802m_User_Data_254_bytes_4_OutputAddress_9 AT %QW1506: WORD;
        st10_is2802m_User_Data_254_bytes_4_OutputAddress_10 AT %QW1508: WORD;
        st10_is2802m_User_Data_254_bytes_4_OutputAddress_11 AT %QW1510: WORD;
        st10_is2802m_User_Data_254_bytes_4_OutputAddress_12 AT %QW1512: WORD;
        st10_is2802m_User_Data_254_bytes_4_OutputAddress_13 AT %QW1514: WORD;
        st10_is2802m_User_Data_254_bytes_4_OutputAddress_14 AT %QW1516: WORD;
        st10_is2802m_User_Data_254_bytes_4_OutputAddress_15 AT %QW1518: WORD;
        st10_is2802m_User_Data_254_bytes_4_OutputAddress_16 AT %QW1520: WORD;
        st10_is2802m_User_Data_254_bytes_4_OutputAddress_17 AT %QW1522: WORD;
        st10_is2802m_User_Data_254_bytes_4_OutputAddress_18 AT %QW1524: WORD;
        st10_is2802m_User_Data_254_bytes_4_OutputAddress_19 AT %QW1526: WORD;
        st10_is2802m_User_Data_254_bytes_4_OutputAddress_20 AT %QW1528: WORD;
        st10_is2802m_User_Data_254_bytes_4_OutputAddress_21 AT %QW1530: WORD;
        st10_is2802m_User_Data_254_bytes_4_OutputAddress_22 AT %QW1532: WORD;
        st10_is2802m_User_Data_254_bytes_4_OutputAddress_23 AT %QW1534: WORD;
        st10_is2802m_User_Data_254_bytes_4_OutputAddress_24 AT %QW1536: WORD;
        st10_is2802m_User_Data_254_bytes_4_OutputAddress_25 AT %QW1538: WORD;
        st10_is2802m_User_Data_254_bytes_4_OutputAddress_26 AT %QW1540: WORD;
        st10_is2802m_User_Data_254_bytes_4_OutputAddress_27 AT %QW1542: WORD;
        st10_is2802m_User_Data_254_bytes_4_OutputAddress_28 AT %QW1544: WORD;
        st10_is2802m_User_Data_254_bytes_4_OutputAddress_29 AT %QW1546: WORD;
        st10_is2802m_User_Data_254_bytes_4_OutputAddress_30 AT %QW1548: WORD;
        st10_is2802m_User_Data_254_bytes_4_OutputAddress_31 AT %QW1550: WORD;
        st10_is2802m_User_Data_254_bytes_4_OutputAddress_32 AT %QW1552: WORD;
        st10_is2802m_User_Data_254_bytes_4_OutputAddress_33 AT %QW1554: WORD;
        st10_is2802m_User_Data_254_bytes_4_OutputAddress_34 AT %QW1556: WORD;
        st10_is2802m_User_Data_254_bytes_4_OutputAddress_35 AT %QW1558: WORD;
        st10_is2802m_User_Data_254_bytes_4_OutputAddress_36 AT %QW1560: WORD;
        st10_is2802m_User_Data_254_bytes_4_OutputAddress_37 AT %QW1562: WORD;
        st10_is2802m_User_Data_254_bytes_4_OutputAddress_38 AT %QW1564: WORD;
        st10_is2802m_User_Data_254_bytes_4_OutputAddress_39 AT %QW1566: WORD;
        st10_is2802m_User_Data_254_bytes_4_OutputAddress_40 AT %QW1568: WORD;
        st10_is2802m_User_Data_254_bytes_4_OutputAddress_41 AT %QW1570: WORD;
        st10_is2802m_User_Data_254_bytes_4_OutputAddress_42 AT %QW1572: WORD;
        st10_is2802m_User_Data_254_bytes_4_OutputAddress_43 AT %QW1574: WORD;
        st10_is2802m_User_Data_254_bytes_4_OutputAddress_44 AT %QW1576: WORD;
        st10_is2802m_User_Data_254_bytes_4_OutputAddress_45 AT %QW1578: WORD;
        st10_is2802m_User_Data_254_bytes_4_OutputAddress_46 AT %QW1580: WORD;
        st10_is2802m_User_Data_254_bytes_4_OutputAddress_47 AT %QW1582: WORD;
        st10_is2802m_User_Data_254_bytes_4_OutputAddress_48 AT %QW1584: WORD;
        st10_is2802m_User_Data_254_bytes_4_OutputAddress_49 AT %QW1586: WORD;
        st10_is2802m_User_Data_254_bytes_4_OutputAddress_50 AT %QW1588: WORD;
        st10_is2802m_User_Data_254_bytes_4_OutputAddress_51 AT %QW1590: WORD;
        st10_is2802m_User_Data_254_bytes_4_OutputAddress_52 AT %QW1592: WORD;
        st10_is2802m_User_Data_254_bytes_4_OutputAddress_53 AT %QW1594: WORD;
        st10_is2802m_User_Data_254_bytes_4_OutputAddress_54 AT %QW1596: WORD;
        st10_is2802m_User_Data_254_bytes_4_OutputAddress_55 AT %QW1598: WORD;
        st10_is2802m_User_Data_254_bytes_4_OutputAddress_56 AT %QW1600: WORD;
        st10_is2802m_User_Data_254_bytes_4_OutputAddress_57 AT %QW1602: WORD;
        st10_is2802m_User_Data_254_bytes_4_OutputAddress_58 AT %QW1604: WORD;
        st10_is2802m_User_Data_254_bytes_4_OutputAddress_59 AT %QW1606: WORD;
        st10_is2802m_User_Data_254_bytes_4_OutputAddress_60 AT %QW1608: WORD;
        st10_is2802m_User_Data_254_bytes_4_OutputAddress_61 AT %QW1610: WORD;
        st10_is2802m_User_Data_254_bytes_4_OutputAddress_62 AT %QW1612: WORD;
        st10_is2802m_User_Data_254_bytes_4_OutputAddress_63 AT %QW1614: WORD;
        st10_is2802m_User_Data_254_bytes_4_OutputAddress_64 AT %QW1616: WORD;
        st10_is2802m_User_Data_254_bytes_4_OutputAddress_65 AT %QW1618: WORD;
        st10_is2802m_User_Data_254_bytes_4_OutputAddress_66 AT %QW1620: WORD;
        st10_is2802m_User_Data_254_bytes_4_OutputAddress_67 AT %QW1622: WORD;
        st10_is2802m_User_Data_254_bytes_4_OutputAddress_68 AT %QW1624: WORD;
        st10_is2802m_User_Data_254_bytes_4_OutputAddress_69 AT %QW1626: WORD;
        st10_is2802m_User_Data_254_bytes_4_OutputAddress_70 AT %QW1628: WORD;
        st10_is2802m_User_Data_254_bytes_4_OutputAddress_71 AT %QW1630: WORD;
        st10_is2802m_User_Data_254_bytes_4_OutputAddress_72 AT %QW1632: WORD;
        st10_is2802m_User_Data_254_bytes_4_OutputAddress_73 AT %QW1634: WORD;
        st10_is2802m_User_Data_254_bytes_4_OutputAddress_74 AT %QW1636: WORD;
        st10_is2802m_User_Data_254_bytes_4_OutputAddress_75 AT %QW1638: WORD;
        st10_is2802m_User_Data_254_bytes_4_OutputAddress_76 AT %QW1640: WORD;
        st10_is2802m_User_Data_254_bytes_4_OutputAddress_77 AT %QW1642: WORD;
        st10_is2802m_User_Data_254_bytes_4_OutputAddress_78 AT %QW1644: WORD;
        st10_is2802m_User_Data_254_bytes_4_OutputAddress_79 AT %QW1646: WORD;
        st10_is2802m_User_Data_254_bytes_4_OutputAddress_80 AT %QW1648: WORD;
        st10_is2802m_User_Data_254_bytes_4_OutputAddress_81 AT %QW1650: WORD;
        st10_is2802m_User_Data_254_bytes_4_OutputAddress_82 AT %QW1652: WORD;
        st10_is2802m_User_Data_254_bytes_4_OutputAddress_83 AT %QW1654: WORD;
        st10_is2802m_User_Data_254_bytes_4_OutputAddress_84 AT %QW1656: WORD;
        st10_is2802m_User_Data_254_bytes_4_OutputAddress_85 AT %QW1658: WORD;
        st10_is2802m_User_Data_254_bytes_4_OutputAddress_86 AT %QW1660: WORD;
        st10_is2802m_User_Data_254_bytes_4_OutputAddress_87 AT %QW1662: WORD;
        st10_is2802m_User_Data_254_bytes_4_OutputAddress_88 AT %QW1664: WORD;
        st10_is2802m_User_Data_254_bytes_4_OutputAddress_89 AT %QW1666: WORD;
        st10_is2802m_User_Data_254_bytes_4_OutputAddress_90 AT %QW1668: WORD;
        st10_is2802m_User_Data_254_bytes_4_OutputAddress_91 AT %QW1670: WORD;
        st10_is2802m_User_Data_254_bytes_4_OutputAddress_92 AT %QW1672: WORD;
        st10_is2802m_User_Data_254_bytes_4_OutputAddress_93 AT %QW1674: WORD;
        st10_is2802m_User_Data_254_bytes_4_OutputAddress_94 AT %QW1676: WORD;
        st10_is2802m_User_Data_254_bytes_4_OutputAddress_95 AT %QW1678: WORD;
        st10_is2802m_User_Data_254_bytes_4_OutputAddress_96 AT %QW1680: WORD;
        st10_is2802m_User_Data_254_bytes_4_OutputAddress_97 AT %QW1682: WORD;
        st10_is2802m_User_Data_254_bytes_4_OutputAddress_98 AT %QW1684: WORD;
        st10_is2802m_User_Data_254_bytes_4_OutputAddress_99 AT %QW1686: WORD;
        st10_is2802m_User_Data_254_bytes_4_OutputAddress_100 AT %QW1688: WORD;
        st10_is2802m_User_Data_254_bytes_4_OutputAddress_101 AT %QW1690: WORD;
        st10_is2802m_User_Data_254_bytes_4_OutputAddress_102 AT %QW1692: WORD;
        st10_is2802m_User_Data_254_bytes_4_OutputAddress_103 AT %QW1694: WORD;
        st10_is2802m_User_Data_254_bytes_4_OutputAddress_104 AT %QW1696: WORD;
        st10_is2802m_User_Data_254_bytes_4_OutputAddress_105 AT %QW1698: WORD;
        st10_is2802m_User_Data_254_bytes_4_OutputAddress_106 AT %QW1700: WORD;
        st10_is2802m_User_Data_254_bytes_4_OutputAddress_107 AT %QW1702: WORD;
        st10_is2802m_User_Data_254_bytes_4_OutputAddress_108 AT %QW1704: WORD;
        st10_is2802m_User_Data_254_bytes_4_OutputAddress_109 AT %QW1706: WORD;
        st10_is2802m_User_Data_254_bytes_4_OutputAddress_110 AT %QW1708: WORD;
        st10_is2802m_User_Data_254_bytes_4_OutputAddress_111 AT %QW1710: WORD;
        st10_is2802m_User_Data_254_bytes_4_OutputAddress_112 AT %QW1712: WORD;
        st10_is2802m_User_Data_254_bytes_4_OutputAddress_113 AT %QW1714: WORD;
        st10_is2802m_User_Data_254_bytes_4_OutputAddress_114 AT %QW1716: WORD;
        st10_is2802m_User_Data_254_bytes_4_OutputAddress_115 AT %QW1718: WORD;
        st10_is2802m_User_Data_254_bytes_4_OutputAddress_116 AT %QW1720: WORD;
        st10_is2802m_User_Data_254_bytes_4_OutputAddress_117 AT %QW1722: WORD;
        st10_is2802m_User_Data_254_bytes_4_OutputAddress_118 AT %QW1724: WORD;
        st10_is2802m_User_Data_254_bytes_4_OutputAddress_119 AT %QW1726: WORD;
        st10_is2802m_User_Data_254_bytes_4_OutputAddress_120 AT %QW1728: WORD;
        st10_is2802m_User_Data_254_bytes_4_OutputAddress_121 AT %QW1730: WORD;
        st10_is2802m_User_Data_254_bytes_4_OutputAddress_122 AT %QW1732: WORD;
        st10_is2802m_User_Data_254_bytes_4_OutputAddress_123 AT %QW1734: WORD;
        st10_is2802m_User_Data_254_bytes_4_OutputAddress_124 AT %QW1736: WORD;
        st10_is2802m_User_Data_254_bytes_4_OutputAddress_125 AT %QW1738: WORD;
        st10_is2802m_User_Data_254_bytes_4_OutputAddress_126 AT %QW1740: WORD;
        st20_is2000_navigation_Acquisition_Control_OutputAddress AT %QB1352: BYTE;
        st20_is2000_navigation_Acquisition_Status_InputAddress_0 AT %IB1384: BYTE;
        st20_is2000_navigation_Acquisition_Status_InputAddress_1 AT %IB1385: BYTE;
        st20_is2000_navigation_Acquisition_Status_InputAddress_2 AT %IB1386: BYTE;
        st20_is2000_navigation_Command_Control_InputAddress AT %IW1387: WORD;
        st20_is2000_navigation_Command_Control_OutputAddress AT %QW1348: WORD;
        st20_is2000_navigation_Inspection_Control_OutputAddress AT %QB1351: BYTE;
        st20_is2000_navigation_Inspection_Status_InputAddress AT %ID1380: DWORD;
        st20_is2000_navigation_Result_Data_64_bytes_InputAddress_0 AT %ID1312: DWORD;
        st20_is2000_navigation_Result_Data_64_bytes_InputAddress_1 AT %ID1316: DWORD;
        st20_is2000_navigation_Result_Data_64_bytes_InputAddress_2 AT %ID1320: DWORD;
        st20_is2000_navigation_Result_Data_64_bytes_InputAddress_3 AT %ID1324: DWORD;
        st20_is2000_navigation_Result_Data_64_bytes_InputAddress_4 AT %ID1328: DWORD;
        st20_is2000_navigation_Result_Data_64_bytes_InputAddress_5 AT %ID1332: DWORD;
        st20_is2000_navigation_Result_Data_64_bytes_InputAddress_6 AT %ID1336: DWORD;
        st20_is2000_navigation_Result_Data_64_bytes_InputAddress_7 AT %ID1340: DWORD;
        st20_is2000_navigation_Result_Data_64_bytes_InputAddress_8 AT %ID1344: DWORD;
        st20_is2000_navigation_Result_Data_64_bytes_InputAddress_9 AT %ID1348: DWORD;
        st20_is2000_navigation_Result_Data_64_bytes_InputAddress_10 AT %ID1352: DWORD;
        st20_is2000_navigation_Result_Data_64_bytes_InputAddress_11 AT %ID1356: DWORD;
        st20_is2000_navigation_Result_Data_64_bytes_InputAddress_12 AT %ID1360: DWORD;
        st20_is2000_navigation_Result_Data_64_bytes_InputAddress_13 AT %ID1364: DWORD;
        st20_is2000_navigation_Result_Data_64_bytes_InputAddress_14 AT %ID1368: DWORD;
        st20_is2000_navigation_Result_Data_64_bytes_InputAddress_15 AT %ID1372: DWORD;
        st20_is2000_navigation_Result_Data_64_bytes_InputAddress_16 AT %ID1376: DWORD;
        st20_is2000_navigation_SoftEvent_Control_InputAddress AT %IB1389: BYTE;
        st20_is2000_navigation_SoftEvent_Control_OutputAddress AT %QB1350: BYTE;
        st20_is2000_navigation_User_Data_64_bytes_OutputAddress_0 AT %QL1284: LWORD;
        st20_is2000_navigation_User_Data_64_bytes_OutputAddress_1 AT %QL1292: LWORD;
        st20_is2000_navigation_User_Data_64_bytes_OutputAddress_2 AT %QL1300: LWORD;
        st20_is2000_navigation_User_Data_64_bytes_OutputAddress_3 AT %QL1308: LWORD;
        st20_is2000_navigation_User_Data_64_bytes_OutputAddress_4 AT %QL1316: LWORD;
        st20_is2000_navigation_User_Data_64_bytes_OutputAddress_5 AT %QL1324: LWORD;
        st20_is2000_navigation_User_Data_64_bytes_OutputAddress_6 AT %QL1332: LWORD;
        st20_is2000_navigation_User_Data_64_bytes_OutputAddress_7 AT %QL1340: LWORD;
